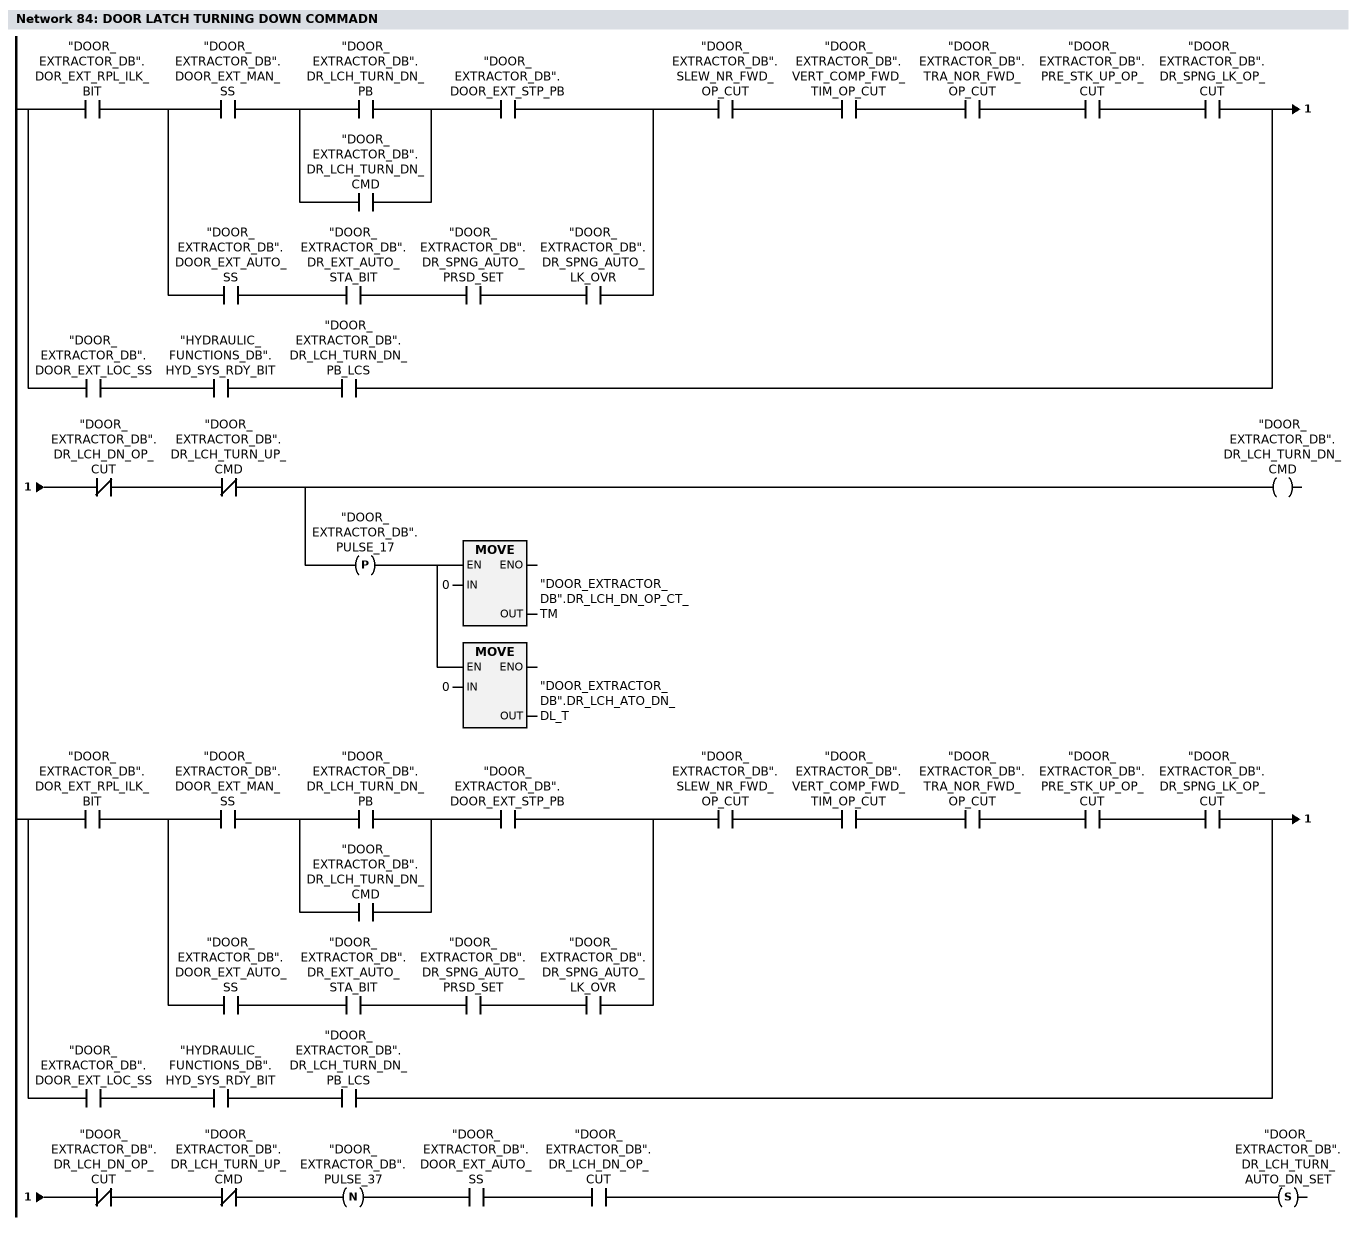
NETWORK
TITLE = DOOR LATCH TURNING DOWN COMMADN
      A(;
      A     "DOOR_EXTRACTOR_DB".DOR_EXT_RPL_ILK_BIT;
      A(;
      A     "DOOR_EXTRACTOR_DB".DOOR_EXT_MAN_SS;
      A(;
      O     "DOOR_EXTRACTOR_DB".DR_LCH_TURN_DN_PB;
      O     "DOOR_EXTRACTOR_DB".DR_LCH_TURN_DN_CMD;
      );
      A     "DOOR_EXTRACTOR_DB".DOOR_EXT_STP_PB;
      O;
      A     "DOOR_EXTRACTOR_DB".DOOR_EXT_AUTO_SS;
      A     "DOOR_EXTRACTOR_DB".DR_EXT_AUTO_STA_BIT;
      A     "DOOR_EXTRACTOR_DB".DR_SPNG_AUTO_PRSD_SET;
      A     "DOOR_EXTRACTOR_DB".DR_SPNG_AUTO_LK_OVR;
      );
      A     "DOOR_EXTRACTOR_DB".SLEW_NR_FWD_OP_CUT;
      A     "DOOR_EXTRACTOR_DB".VERT_COMP_FWD_TIM_OP_CUT;
      A     "DOOR_EXTRACTOR_DB".TRA_NOR_FWD_OP_CUT;
      A     "DOOR_EXTRACTOR_DB".PRE_STK_UP_OP_CUT;
      A     "DOOR_EXTRACTOR_DB".DR_SPNG_LK_OP_CUT;
      O;
      A     "DOOR_EXTRACTOR_DB".DOOR_EXT_LOC_SS;
      A     "HYDRAULIC_FUNCTIONS_DB".HYD_SYS_RDY_BIT;
      A     "DOOR_EXTRACTOR_DB".DR_LCH_TURN_DN_PB_LCS;
      );
      AN    "DOOR_EXTRACTOR_DB".DR_LCH_DN_OP_CUT;
      AN    "DOOR_EXTRACTOR_DB".DR_LCH_TURN_UP_CMD;
      =     L 0.0;
      A     L 0.0;
      BLD   102;
      =     "DOOR_EXTRACTOR_DB".DR_LCH_TURN_DN_CMD;
      A(;
      A     L 0.0;
      FN    "DOOR_EXTRACTOR_DB".PULSE_37;
      );
      A     "DOOR_EXTRACTOR_DB".DOOR_EXT_AUTO_SS;
      A     "DOOR_EXTRACTOR_DB".DR_LCH_DN_OP_CUT;
      S     "DOOR_EXTRACTOR_DB".DR_LCH_TURN_AUTO_DN_SET;
      A     L 0.0;
      FP    "DOOR_EXTRACTOR_DB".PULSE_17;
      =     L 0.1;
      A     L 0.1;
      JNB   _04b;
      L     0;
      T     "DOOR_EXTRACTOR_DB".DR_LCH_DN_OP_CT_TM;
_04b: NOP   0;
      A     L 0.1;
      JNB   _04c;
      L     0;
      T     "DOOR_EXTRACTOR_DB".DR_LCH_ATO_DN_DL_T;
_04c: NOP   0;
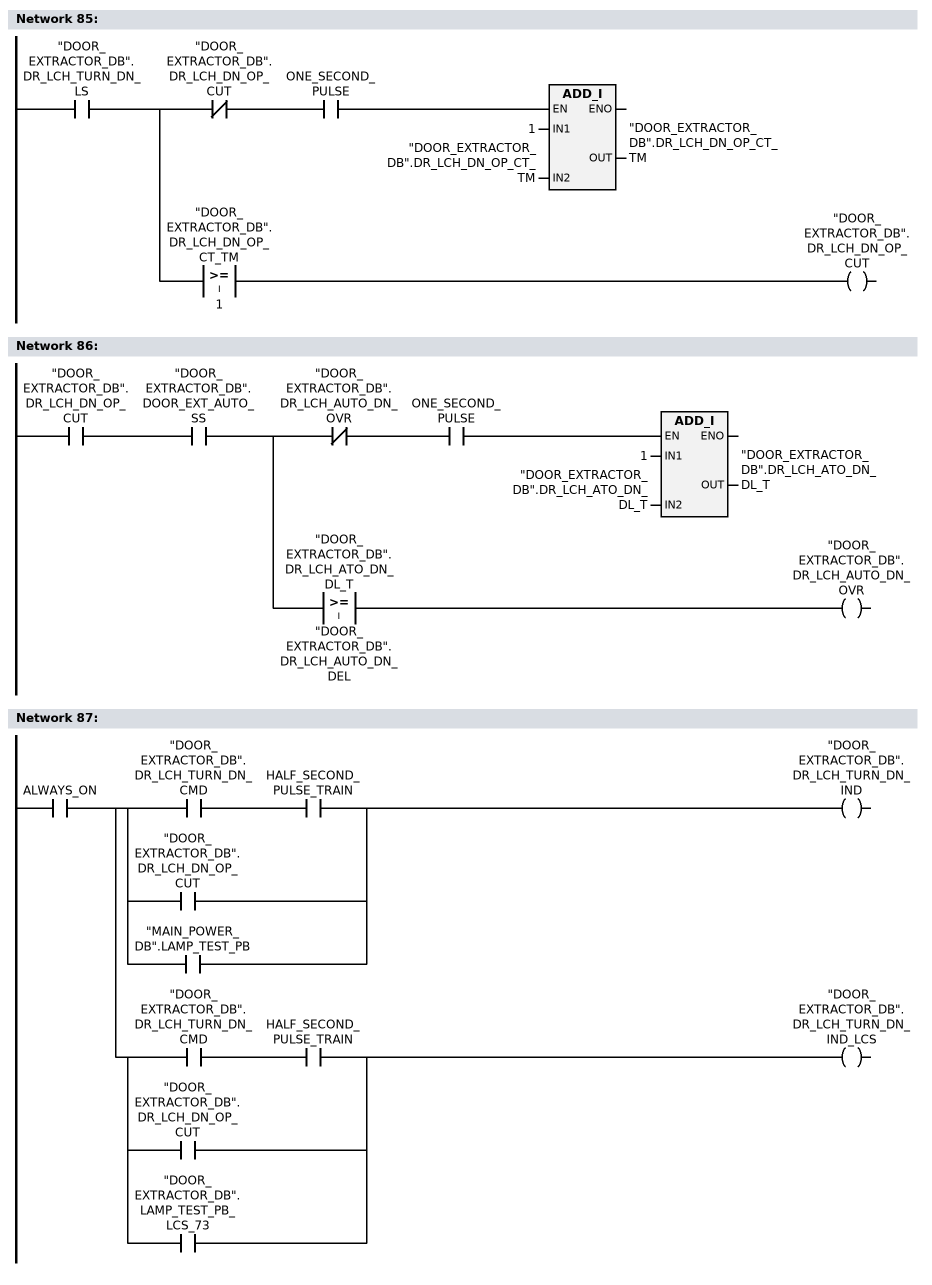
NETWORK
TITLE =
      A     "DOOR_EXTRACTOR_DB".DR_LCH_TURN_DN_LS;
      =     L 0.0;
      A     L 0.0;
      AN    "DOOR_EXTRACTOR_DB".DR_LCH_DN_OP_CUT;
      A     "ONE_SECOND_PULSE";
      JNB   _04d;
      L     1;
      L     "DOOR_EXTRACTOR_DB".DR_LCH_DN_OP_CT_TM;
      +I;
      T     "DOOR_EXTRACTOR_DB".DR_LCH_DN_OP_CT_TM;
_04d: NOP   0;
      A     L 0.0;
      A(;
      L     "DOOR_EXTRACTOR_DB".DR_LCH_DN_OP_CT_TM;
      L     1;
      >=I;
      );
      =     "DOOR_EXTRACTOR_DB".DR_LCH_DN_OP_CUT;
NETWORK
TITLE =
      A     "DOOR_EXTRACTOR_DB".DR_LCH_DN_OP_CUT;
      A     "DOOR_EXTRACTOR_DB".DOOR_EXT_AUTO_SS;
      =     L 0.0;
      A     L 0.0;
      AN    "DOOR_EXTRACTOR_DB".DR_LCH_AUTO_DN_OVR;
      A     "ONE_SECOND_PULSE";
      JNB   _04e;
      L     1;
      L     "DOOR_EXTRACTOR_DB".DR_LCH_ATO_DN_DL_T;
      +I;
      T     "DOOR_EXTRACTOR_DB".DR_LCH_ATO_DN_DL_T;
_04e: NOP   0;
      A     L 0.0;
      A(;
      L     "DOOR_EXTRACTOR_DB".DR_LCH_ATO_DN_DL_T;
      L     "DOOR_EXTRACTOR_DB".DR_LCH_AUTO_DN_DEL;
      >=I;
      );
      =     "DOOR_EXTRACTOR_DB".DR_LCH_AUTO_DN_OVR;
NETWORK
TITLE =
      A     "ALWAYS_ON";
      =     L 0.0;
      A     L 0.0;
      A(;
      A     "DOOR_EXTRACTOR_DB".DR_LCH_TURN_DN_CMD;
      A     "HALF_SECOND_PULSE_TRAIN";
      O     "DOOR_EXTRACTOR_DB".DR_LCH_DN_OP_CUT;
      O     "MAIN_POWER_DB".LAMP_TEST_PB;
      );
      =     "DOOR_EXTRACTOR_DB".DR_LCH_TURN_DN_IND;
      A     L 0.0;
      A(;
      A     "DOOR_EXTRACTOR_DB".DR_LCH_TURN_DN_CMD;
      A     "HALF_SECOND_PULSE_TRAIN";
      O     "DOOR_EXTRACTOR_DB".DR_LCH_DN_OP_CUT;
      O     "DOOR_EXTRACTOR_DB".LAMP_TEST_PB_LCS_73;
      );
      =     "DOOR_EXTRACTOR_DB".DR_LCH_TURN_DN_IND_LCS;
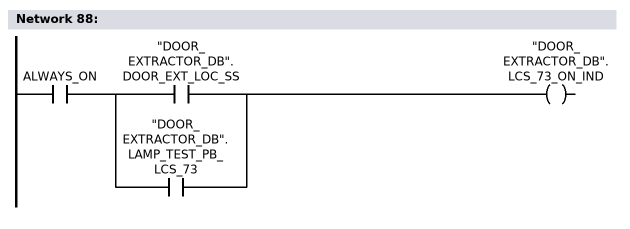
NETWORK
TITLE =
      A     "ALWAYS_ON";
      A(;
      O     "DOOR_EXTRACTOR_DB".DOOR_EXT_LOC_SS;
      O     "DOOR_EXTRACTOR_DB".LAMP_TEST_PB_LCS_73;
      );
      =     "DOOR_EXTRACTOR_DB".LCS_73_ON_IND;
END_FUNCTION

FUNCTION "DOOR_CLEANER" : VOID	// FC 15
AUTHOR : Kamillas
VERSION : 0.1
BEGIN
// (block stored without names or comments; labels and parameter names are numbered)
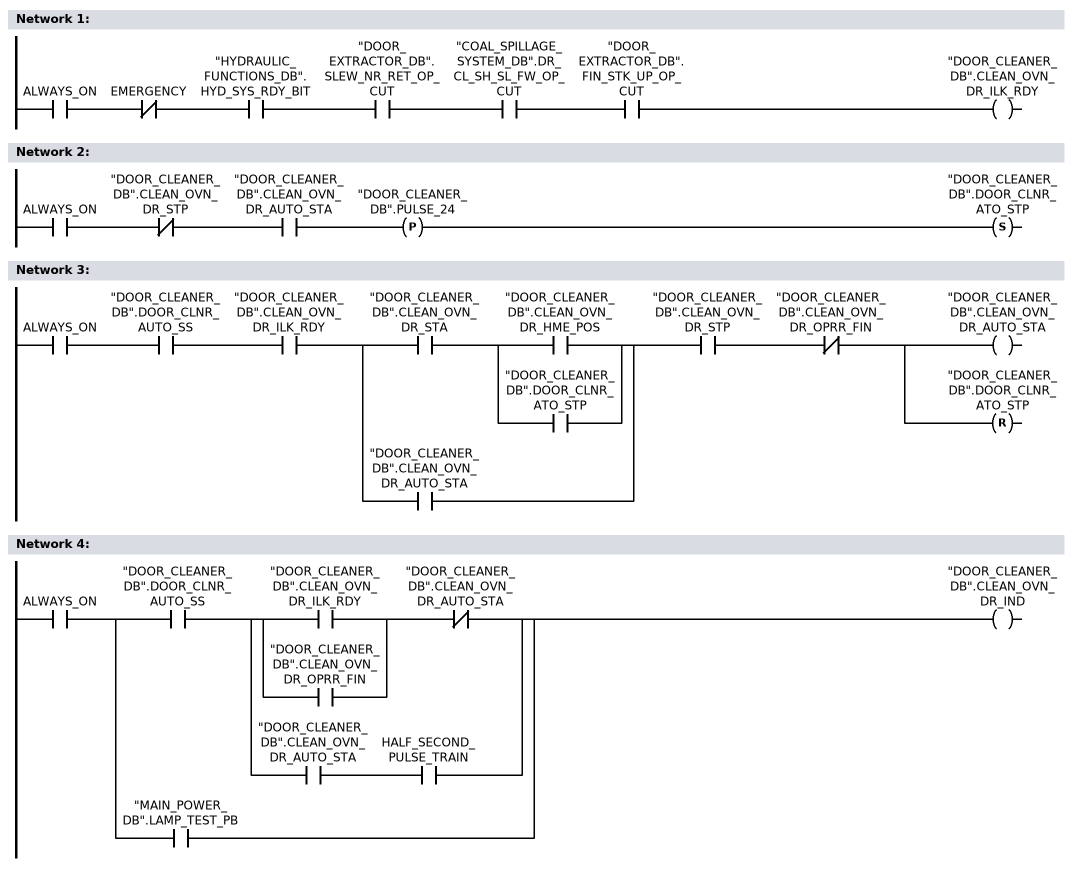
NETWORK
TITLE =
      A     "ALWAYS_ON";
      AN    "EMERGENCY";
      A     "HYDRAULIC_FUNCTIONS_DB".HYD_SYS_RDY_BIT;
      A     "DOOR_EXTRACTOR_DB".SLEW_NR_RET_OP_CUT;
      A     "COAL_SPILLAGE_SYSTEM_DB".DR_CL_SH_SL_FW_OP_CUT;
      A     "DOOR_EXTRACTOR_DB".FIN_STK_UP_OP_CUT;
      =     "DOOR_CLEANER_DB".CLEAN_OVN_DR_ILK_RDY;
NETWORK
TITLE =
      A     "ALWAYS_ON";
      AN    "DOOR_CLEANER_DB".CLEAN_OVN_DR_STP;
      A     "DOOR_CLEANER_DB".CLEAN_OVN_DR_AUTO_STA;
      FP    "DOOR_CLEANER_DB".PULSE_24;
      S     "DOOR_CLEANER_DB".DOOR_CLNR_ATO_STP;
NETWORK
TITLE =
      A     "ALWAYS_ON";
      A     "DOOR_CLEANER_DB".DOOR_CLNR_AUTO_SS;
      A     "DOOR_CLEANER_DB".CLEAN_OVN_DR_ILK_RDY;
      A(;
      A     "DOOR_CLEANER_DB".CLEAN_OVN_DR_STA;
      A(;
      O     "DOOR_CLEANER_DB".CLEAN_OVN_DR_HME_POS;
      O     "DOOR_CLEANER_DB".DOOR_CLNR_ATO_STP;
      );
      O     "DOOR_CLEANER_DB".CLEAN_OVN_DR_AUTO_STA;
      );
      A     "DOOR_CLEANER_DB".CLEAN_OVN_DR_STP;
      AN    "DOOR_CLEANER_DB".CLEAN_OVN_DR_OPRR_FIN;
      =     "DOOR_CLEANER_DB".CLEAN_OVN_DR_AUTO_STA;
      R     "DOOR_CLEANER_DB".DOOR_CLNR_ATO_STP;
NETWORK
TITLE =
      A     "ALWAYS_ON";
      A(;
      A     "DOOR_CLEANER_DB".DOOR_CLNR_AUTO_SS;
      A(;
      A(;
      O     "DOOR_CLEANER_DB".CLEAN_OVN_DR_ILK_RDY;
      O     "DOOR_CLEANER_DB".CLEAN_OVN_DR_OPRR_FIN;
      );
      AN    "DOOR_CLEANER_DB".CLEAN_OVN_DR_AUTO_STA;
      O;
      A     "DOOR_CLEANER_DB".CLEAN_OVN_DR_AUTO_STA;
      A     "HALF_SECOND_PULSE_TRAIN";
      );
      O     "MAIN_POWER_DB".LAMP_TEST_PB;
      );
      =     "DOOR_CLEANER_DB".CLEAN_OVN_DR_IND;
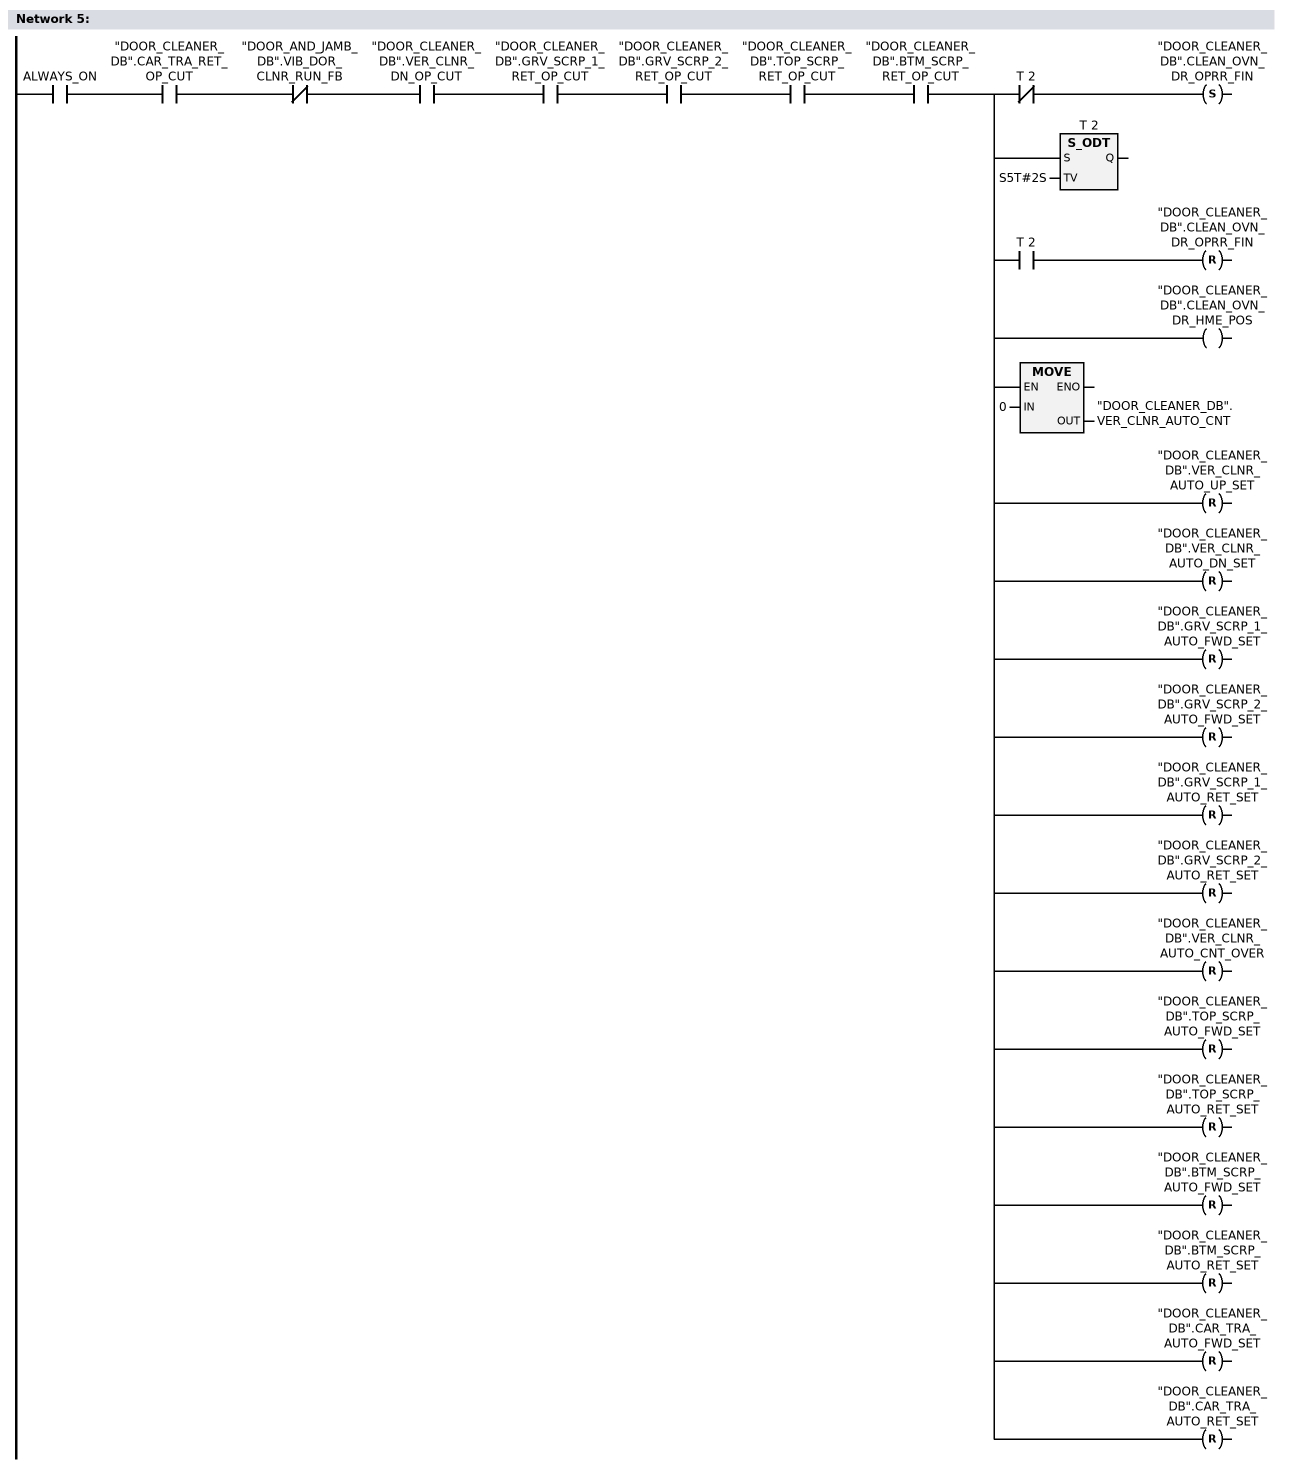
NETWORK
TITLE =
      A     "ALWAYS_ON";
      A     "DOOR_CLEANER_DB".CAR_TRA_RET_OP_CUT;
      AN    "DOOR_AND_JAMB_DB".VIB_DOR_CLNR_RUN_FB;
      A     "DOOR_CLEANER_DB".VER_CLNR_DN_OP_CUT;
      A     "DOOR_CLEANER_DB".GRV_SCRP_1_RET_OP_CUT;
      A     "DOOR_CLEANER_DB".GRV_SCRP_2_RET_OP_CUT;
      A     "DOOR_CLEANER_DB".TOP_SCRP_RET_OP_CUT;
      A     "DOOR_CLEANER_DB".BTM_SCRP_RET_OP_CUT;
      =     L 0.0;
      A     L 0.0;
      AN    T 2;
      S     "DOOR_CLEANER_DB".CLEAN_OVN_DR_OPRR_FIN;
      A     L 0.0;
      L     S5T#2S;
      SD    T 2;
      NOP   0;
      NOP   0;
      NOP   0;
      NOP   0;
      A     L 0.0;
      A     T 2;
      R     "DOOR_CLEANER_DB".CLEAN_OVN_DR_OPRR_FIN;
      A     L 0.0;
      BLD   102;
      =     "DOOR_CLEANER_DB".CLEAN_OVN_DR_HME_POS;
      A     L 0.0;
      JNB   M001;
      L     0;
      T     "DOOR_CLEANER_DB".VER_CLNR_AUTO_CNT;
M001: NOP   0;
      A     L 0.0;
      BLD   102;
      R     "DOOR_CLEANER_DB".VER_CLNR_AUTO_UP_SET;
      A     L 0.0;
      BLD   102;
      R     "DOOR_CLEANER_DB".VER_CLNR_AUTO_DN_SET;
      A     L 0.0;
      BLD   102;
      R     "DOOR_CLEANER_DB".GRV_SCRP_1_AUTO_FWD_SET;
      A     L 0.0;
      BLD   102;
      R     "DOOR_CLEANER_DB".GRV_SCRP_2_AUTO_FWD_SET;
      A     L 0.0;
      BLD   102;
      R     "DOOR_CLEANER_DB".GRV_SCRP_1_AUTO_RET_SET;
      A     L 0.0;
      BLD   102;
      R     "DOOR_CLEANER_DB".GRV_SCRP_2_AUTO_RET_SET;
      A     L 0.0;
      BLD   102;
      R     "DOOR_CLEANER_DB".VER_CLNR_AUTO_CNT_OVER;
      A     L 0.0;
      BLD   102;
      R     "DOOR_CLEANER_DB".TOP_SCRP_AUTO_FWD_SET;
      A     L 0.0;
      BLD   102;
      R     "DOOR_CLEANER_DB".TOP_SCRP_AUTO_RET_SET;
      A     L 0.0;
      BLD   102;
      R     "DOOR_CLEANER_DB".BTM_SCRP_AUTO_FWD_SET;
      A     L 0.0;
      BLD   102;
      R     "DOOR_CLEANER_DB".BTM_SCRP_AUTO_RET_SET;
      A     L 0.0;
      BLD   102;
      R     "DOOR_CLEANER_DB".CAR_TRA_AUTO_FWD_SET;
      A     L 0.0;
      BLD   102;
      R     "DOOR_CLEANER_DB".CAR_TRA_AUTO_RET_SET;
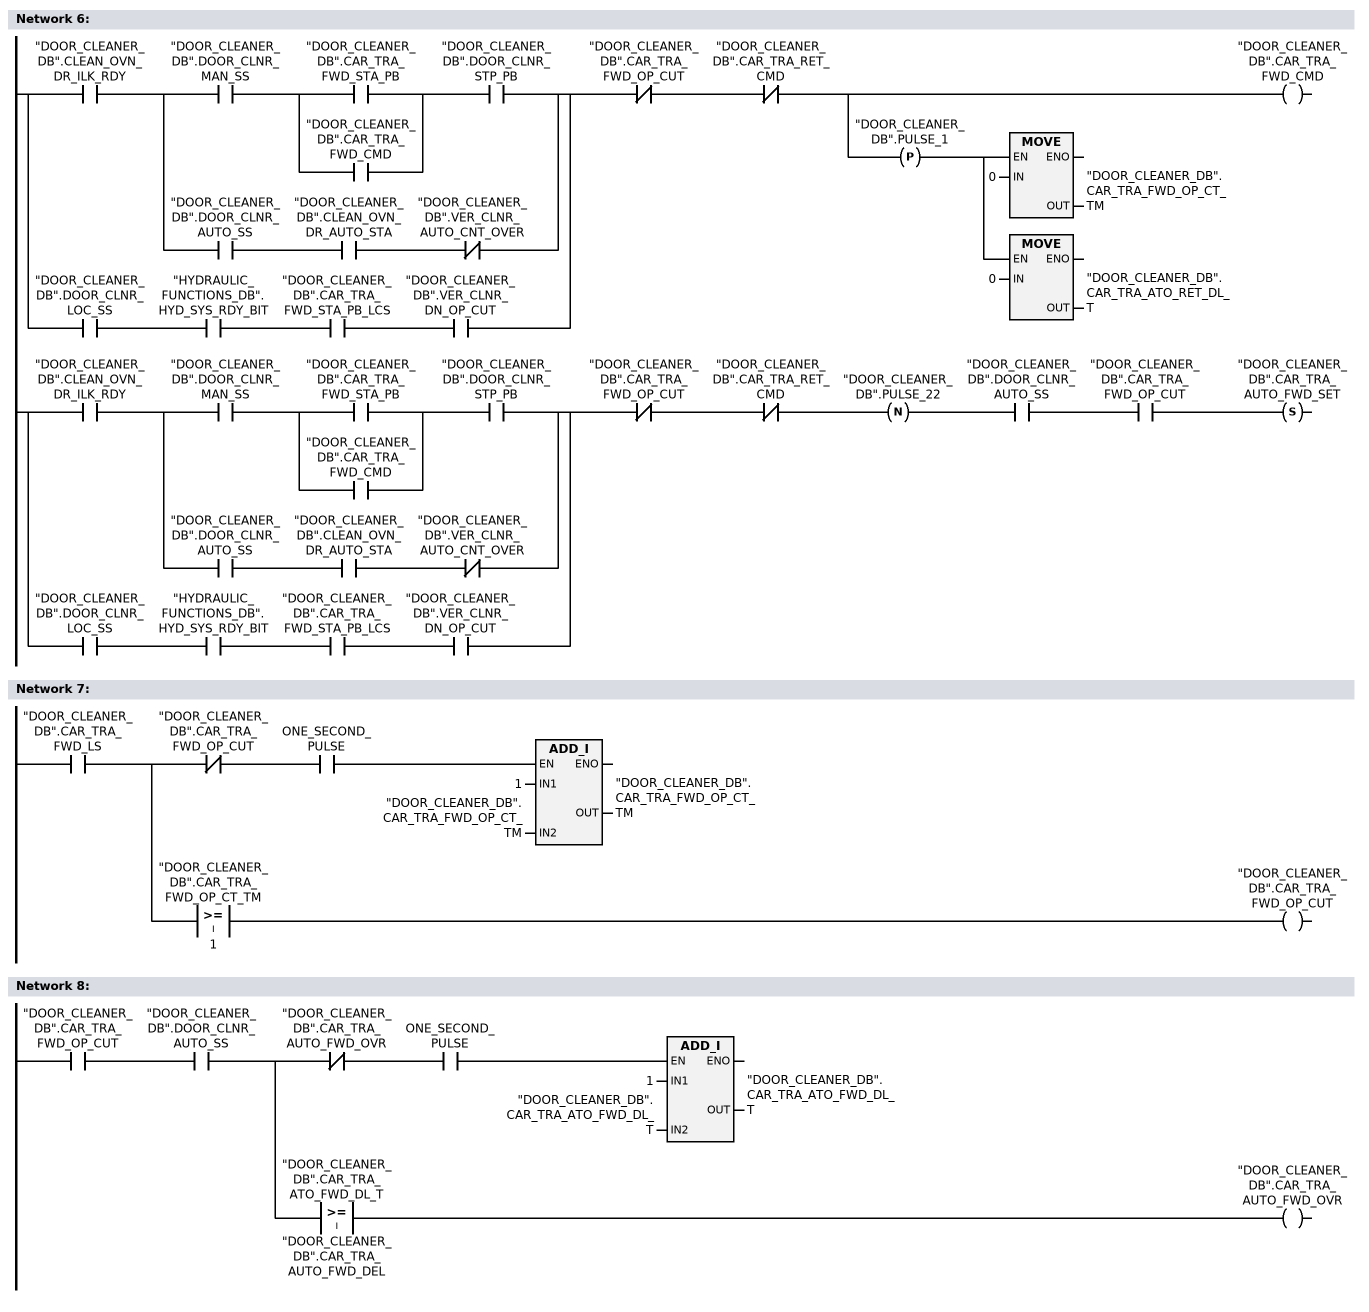
NETWORK
TITLE =
      A(;
      A     "DOOR_CLEANER_DB".CLEAN_OVN_DR_ILK_RDY;
      A(;
      A     "DOOR_CLEANER_DB".DOOR_CLNR_MAN_SS;
      A(;
      O     "DOOR_CLEANER_DB".CAR_TRA_FWD_STA_PB;
      O     "DOOR_CLEANER_DB".CAR_TRA_FWD_CMD;
      );
      A     "DOOR_CLEANER_DB".DOOR_CLNR_STP_PB;
      O;
      A     "DOOR_CLEANER_DB".DOOR_CLNR_AUTO_SS;
      A     "DOOR_CLEANER_DB".CLEAN_OVN_DR_AUTO_STA;
      AN    "DOOR_CLEANER_DB".VER_CLNR_AUTO_CNT_OVER;
      );
      O;
      A     "DOOR_CLEANER_DB".DOOR_CLNR_LOC_SS;
      A     "HYDRAULIC_FUNCTIONS_DB".HYD_SYS_RDY_BIT;
      A     "DOOR_CLEANER_DB".CAR_TRA_FWD_STA_PB_LCS;
      A     "DOOR_CLEANER_DB".VER_CLNR_DN_OP_CUT;
      );
      AN    "DOOR_CLEANER_DB".CAR_TRA_FWD_OP_CUT;
      AN    "DOOR_CLEANER_DB".CAR_TRA_RET_CMD;
      =     L 0.0;
      A     L 0.0;
      BLD   102;
      =     "DOOR_CLEANER_DB".CAR_TRA_FWD_CMD;
      A(;
      A     L 0.0;
      FN    "DOOR_CLEANER_DB".PULSE_22;
      );
      A     "DOOR_CLEANER_DB".DOOR_CLNR_AUTO_SS;
      A     "DOOR_CLEANER_DB".CAR_TRA_FWD_OP_CUT;
      S     "DOOR_CLEANER_DB".CAR_TRA_AUTO_FWD_SET;
      A     L 0.0;
      FP    "DOOR_CLEANER_DB".PULSE_1;
      =     L 0.1;
      A     L 0.1;
      JNB   M002;
      L     0;
      T     "DOOR_CLEANER_DB".CAR_TRA_FWD_OP_CT_TM;
M002: NOP   0;
      A     L 0.1;
      JNB   M003;
      L     0;
      T     "DOOR_CLEANER_DB".CAR_TRA_ATO_RET_DL_T;
M003: NOP   0;
NETWORK
TITLE =
      A     "DOOR_CLEANER_DB".CAR_TRA_FWD_LS;
      =     L 0.0;
      A     L 0.0;
      AN    "DOOR_CLEANER_DB".CAR_TRA_FWD_OP_CUT;
      A     "ONE_SECOND_PULSE";
      JNB   M004;
      L     1;
      L     "DOOR_CLEANER_DB".CAR_TRA_FWD_OP_CT_TM;
      +I;
      T     "DOOR_CLEANER_DB".CAR_TRA_FWD_OP_CT_TM;
M004: NOP   0;
      A     L 0.0;
      A(;
      L     "DOOR_CLEANER_DB".CAR_TRA_FWD_OP_CT_TM;
      L     1;
      >=I;
      );
      =     "DOOR_CLEANER_DB".CAR_TRA_FWD_OP_CUT;
NETWORK
TITLE =
      A     "DOOR_CLEANER_DB".CAR_TRA_FWD_OP_CUT;
      A     "DOOR_CLEANER_DB".DOOR_CLNR_AUTO_SS;
      =     L 0.0;
      A     L 0.0;
      AN    "DOOR_CLEANER_DB".CAR_TRA_AUTO_FWD_OVR;
      A     "ONE_SECOND_PULSE";
      JNB   M005;
      L     1;
      L     "DOOR_CLEANER_DB".CAR_TRA_ATO_FWD_DL_T;
      +I;
      T     "DOOR_CLEANER_DB".CAR_TRA_ATO_FWD_DL_T;
M005: NOP   0;
      A     L 0.0;
      A(;
      L     "DOOR_CLEANER_DB".CAR_TRA_ATO_FWD_DL_T;
      L     "DOOR_CLEANER_DB".CAR_TRA_AUTO_FWD_DEL;
      >=I;
      );
      =     "DOOR_CLEANER_DB".CAR_TRA_AUTO_FWD_OVR;
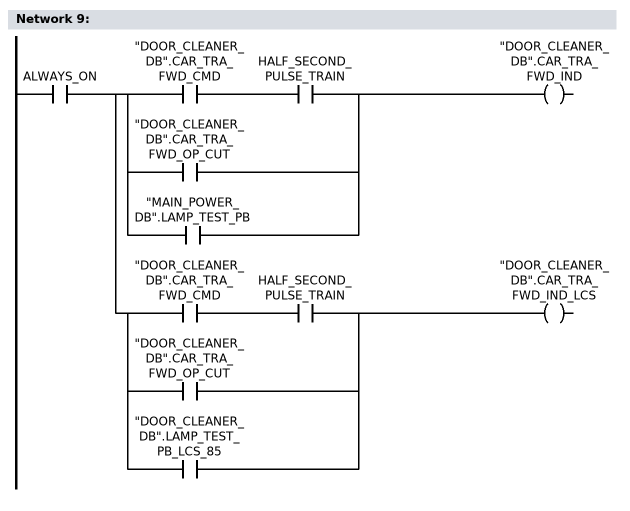
NETWORK
TITLE =
      A     "ALWAYS_ON";
      =     L 0.0;
      A     L 0.0;
      A(;
      A     "DOOR_CLEANER_DB".CAR_TRA_FWD_CMD;
      A     "HALF_SECOND_PULSE_TRAIN";
      O     "DOOR_CLEANER_DB".CAR_TRA_FWD_OP_CUT;
      O     "MAIN_POWER_DB".LAMP_TEST_PB;
      );
      =     "DOOR_CLEANER_DB".CAR_TRA_FWD_IND;
      A     L 0.0;
      A(;
      A     "DOOR_CLEANER_DB".CAR_TRA_FWD_CMD;
      A     "HALF_SECOND_PULSE_TRAIN";
      O     "DOOR_CLEANER_DB".CAR_TRA_FWD_OP_CUT;
      O     "DOOR_CLEANER_DB".LAMP_TEST_PB_LCS_85;
      );
      =     "DOOR_CLEANER_DB".CAR_TRA_FWD_IND_LCS;
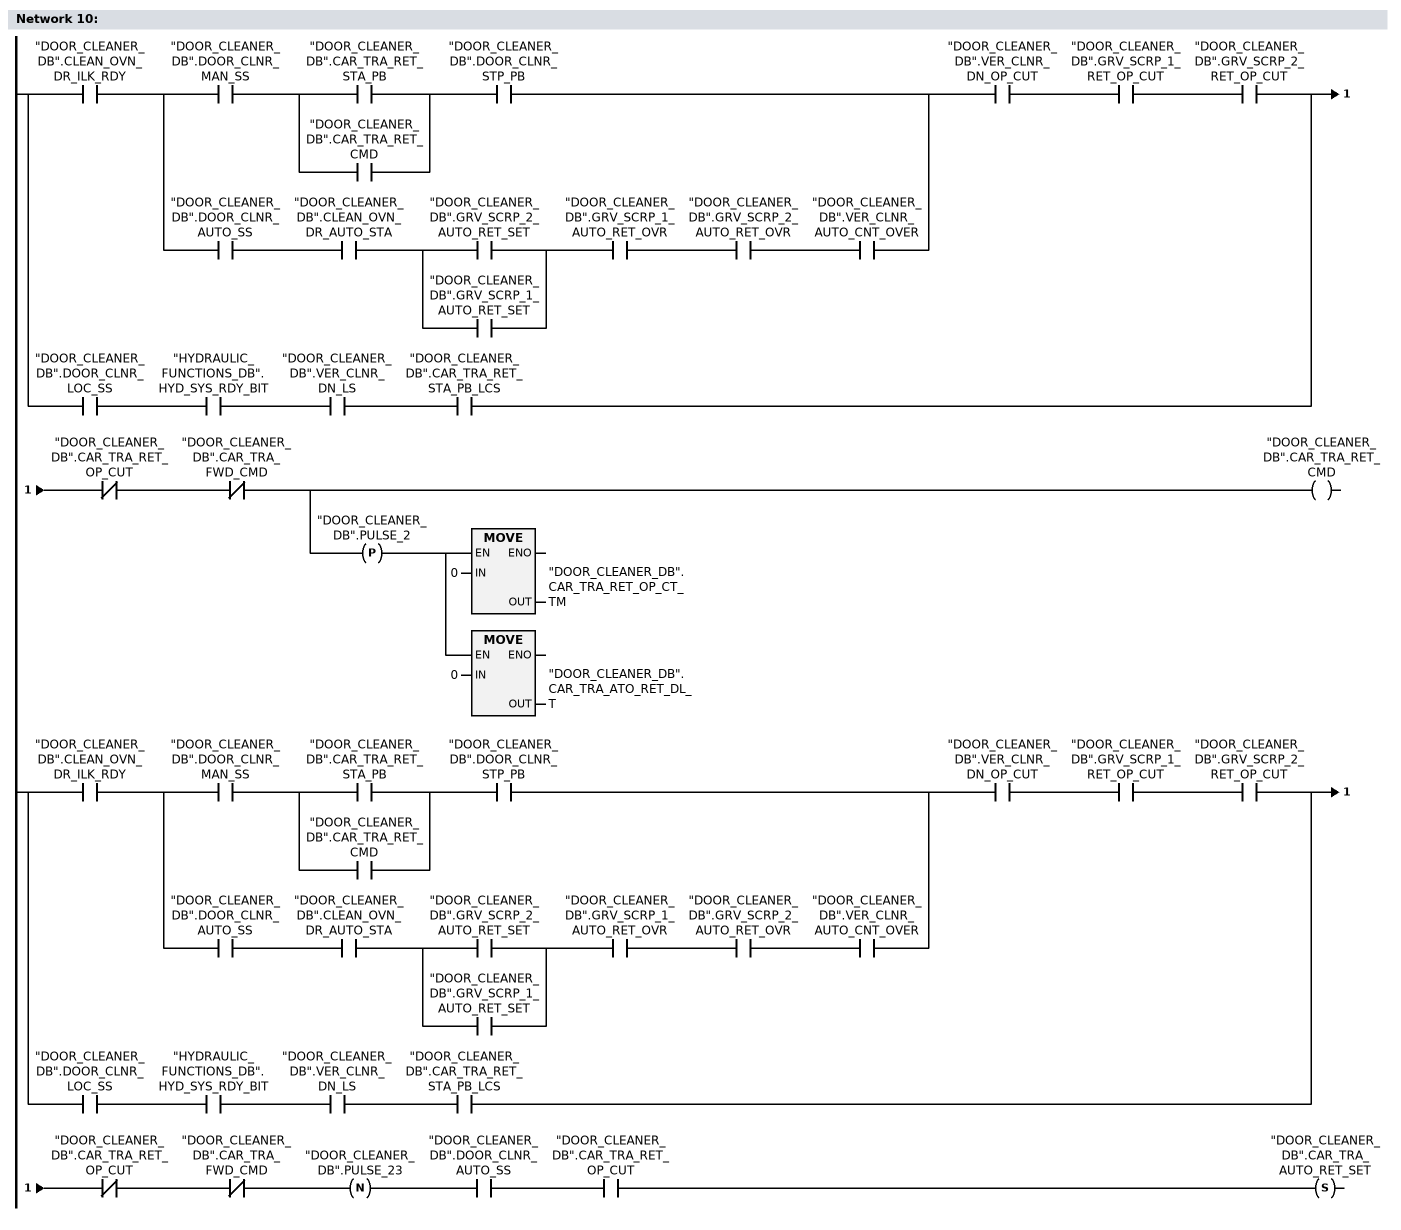
NETWORK
TITLE =
      A(;
      A     "DOOR_CLEANER_DB".CLEAN_OVN_DR_ILK_RDY;
      A(;
      A     "DOOR_CLEANER_DB".DOOR_CLNR_MAN_SS;
      A(;
      O     "DOOR_CLEANER_DB".CAR_TRA_RET_STA_PB;
      O     "DOOR_CLEANER_DB".CAR_TRA_RET_CMD;
      );
      A     "DOOR_CLEANER_DB".DOOR_CLNR_STP_PB;
      O;
      A     "DOOR_CLEANER_DB".DOOR_CLNR_AUTO_SS;
      A     "DOOR_CLEANER_DB".CLEAN_OVN_DR_AUTO_STA;
      A(;
      O     "DOOR_CLEANER_DB".GRV_SCRP_2_AUTO_RET_SET;
      O     "DOOR_CLEANER_DB".GRV_SCRP_1_AUTO_RET_SET;
      );
      A     "DOOR_CLEANER_DB".GRV_SCRP_1_AUTO_RET_OVR;
      A     "DOOR_CLEANER_DB".GRV_SCRP_2_AUTO_RET_OVR;
      A     "DOOR_CLEANER_DB".VER_CLNR_AUTO_CNT_OVER;
      );
      A     "DOOR_CLEANER_DB".VER_CLNR_DN_OP_CUT;
      A     "DOOR_CLEANER_DB".GRV_SCRP_1_RET_OP_CUT;
      A     "DOOR_CLEANER_DB".GRV_SCRP_2_RET_OP_CUT;
      O;
      A     "DOOR_CLEANER_DB".DOOR_CLNR_LOC_SS;
      A     "HYDRAULIC_FUNCTIONS_DB".HYD_SYS_RDY_BIT;
      A     "DOOR_CLEANER_DB".VER_CLNR_DN_LS;
      A     "DOOR_CLEANER_DB".CAR_TRA_RET_STA_PB_LCS;
      );
      AN    "DOOR_CLEANER_DB".CAR_TRA_RET_OP_CUT;
      AN    "DOOR_CLEANER_DB".CAR_TRA_FWD_CMD;
      =     L 0.0;
      A     L 0.0;
      BLD   102;
      =     "DOOR_CLEANER_DB".CAR_TRA_RET_CMD;
      A(;
      A     L 0.0;
      FN    "DOOR_CLEANER_DB".PULSE_23;
      );
      A     "DOOR_CLEANER_DB".DOOR_CLNR_AUTO_SS;
      A     "DOOR_CLEANER_DB".CAR_TRA_RET_OP_CUT;
      S     "DOOR_CLEANER_DB".CAR_TRA_AUTO_RET_SET;
      A     L 0.0;
      FP    "DOOR_CLEANER_DB".PULSE_2;
      =     L 0.1;
      A     L 0.1;
      JNB   M006;
      L     0;
      T     "DOOR_CLEANER_DB".CAR_TRA_RET_OP_CT_TM;
M006: NOP   0;
      A     L 0.1;
      JNB   M007;
      L     0;
      T     "DOOR_CLEANER_DB".CAR_TRA_ATO_RET_DL_T;
M007: NOP   0;
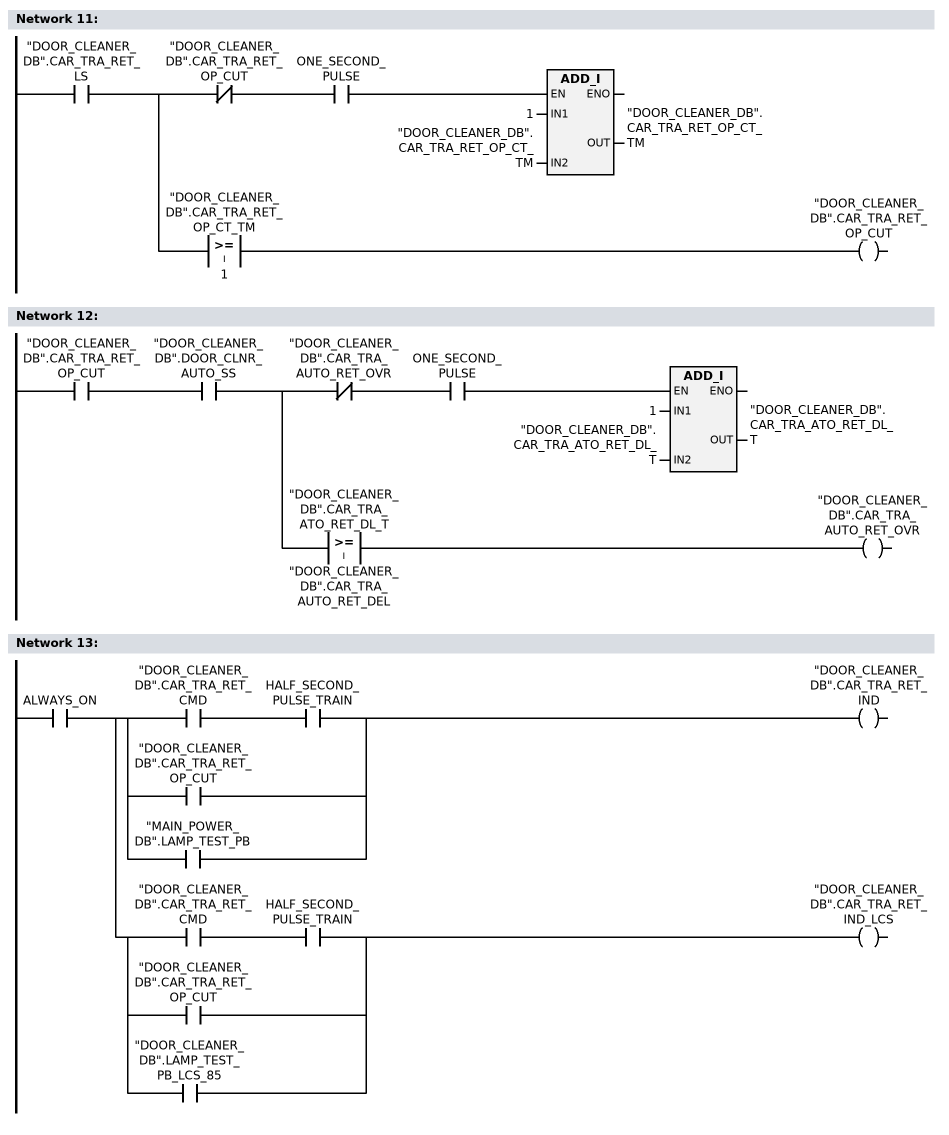
NETWORK
TITLE =
      A     "DOOR_CLEANER_DB".CAR_TRA_RET_LS;
      =     L 0.0;
      A     L 0.0;
      AN    "DOOR_CLEANER_DB".CAR_TRA_RET_OP_CUT;
      A     "ONE_SECOND_PULSE";
      JNB   M008;
      L     1;
      L     "DOOR_CLEANER_DB".CAR_TRA_RET_OP_CT_TM;
      +I;
      T     "DOOR_CLEANER_DB".CAR_TRA_RET_OP_CT_TM;
M008: NOP   0;
      A     L 0.0;
      A(;
      L     "DOOR_CLEANER_DB".CAR_TRA_RET_OP_CT_TM;
      L     1;
      >=I;
      );
      =     "DOOR_CLEANER_DB".CAR_TRA_RET_OP_CUT;
NETWORK
TITLE =
      A     "DOOR_CLEANER_DB".CAR_TRA_RET_OP_CUT;
      A     "DOOR_CLEANER_DB".DOOR_CLNR_AUTO_SS;
      =     L 0.0;
      A     L 0.0;
      AN    "DOOR_CLEANER_DB".CAR_TRA_AUTO_RET_OVR;
      A     "ONE_SECOND_PULSE";
      JNB   M009;
      L     1;
      L     "DOOR_CLEANER_DB".CAR_TRA_ATO_RET_DL_T;
      +I;
      T     "DOOR_CLEANER_DB".CAR_TRA_ATO_RET_DL_T;
M009: NOP   0;
      A     L 0.0;
      A(;
      L     "DOOR_CLEANER_DB".CAR_TRA_ATO_RET_DL_T;
      L     "DOOR_CLEANER_DB".CAR_TRA_AUTO_RET_DEL;
      >=I;
      );
      =     "DOOR_CLEANER_DB".CAR_TRA_AUTO_RET_OVR;
NETWORK
TITLE =
      A     "ALWAYS_ON";
      =     L 0.0;
      A     L 0.0;
      A(;
      A     "DOOR_CLEANER_DB".CAR_TRA_RET_CMD;
      A     "HALF_SECOND_PULSE_TRAIN";
      O     "DOOR_CLEANER_DB".CAR_TRA_RET_OP_CUT;
      O     "MAIN_POWER_DB".LAMP_TEST_PB;
      );
      =     "DOOR_CLEANER_DB".CAR_TRA_RET_IND;
      A     L 0.0;
      A(;
      A     "DOOR_CLEANER_DB".CAR_TRA_RET_CMD;
      A     "HALF_SECOND_PULSE_TRAIN";
      O     "DOOR_CLEANER_DB".CAR_TRA_RET_OP_CUT;
      O     "DOOR_CLEANER_DB".LAMP_TEST_PB_LCS_85;
      );
      =     "DOOR_CLEANER_DB".CAR_TRA_RET_IND_LCS;
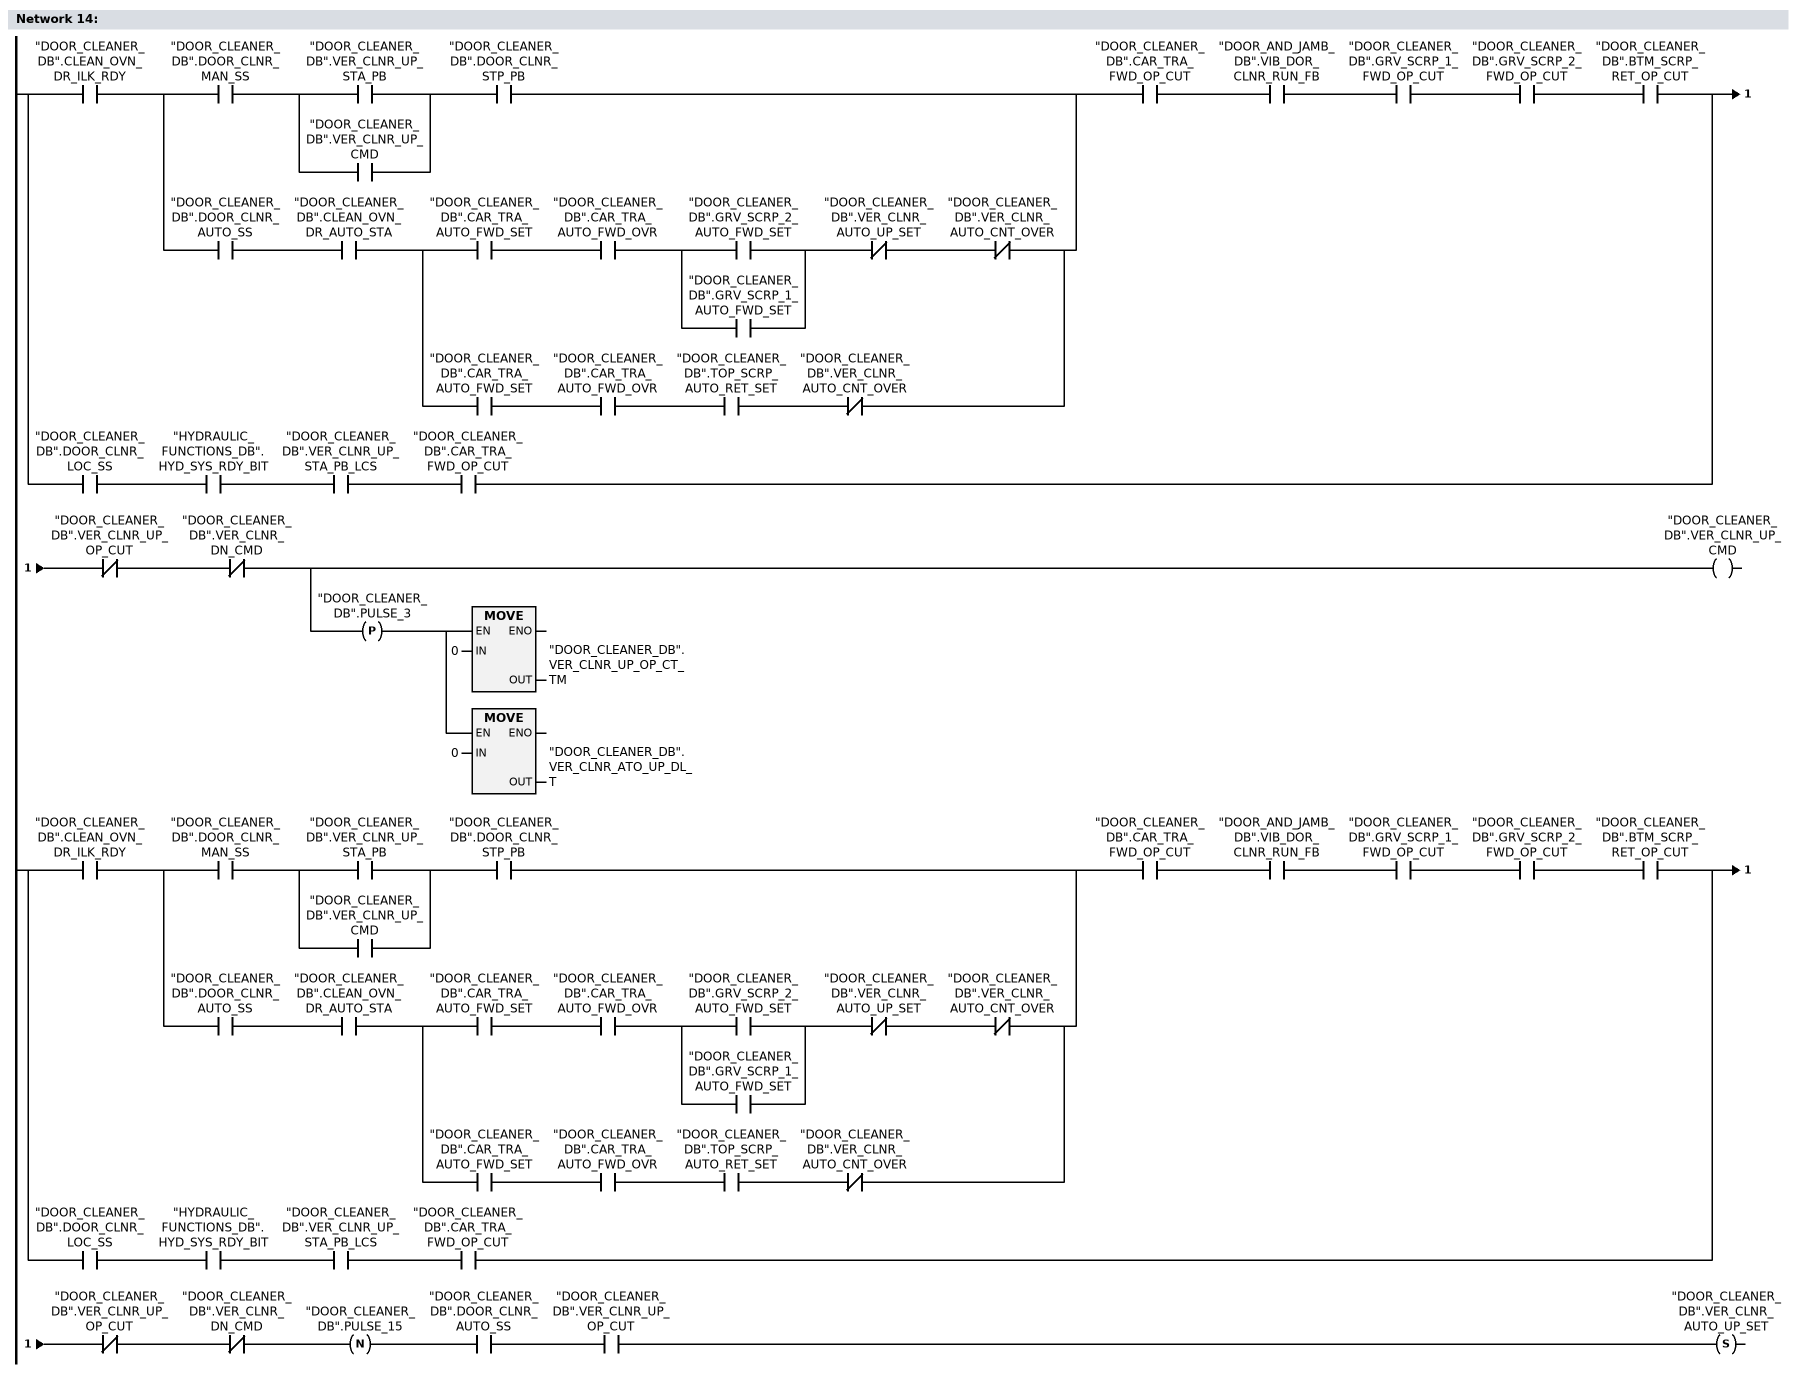
NETWORK
TITLE =
      A(;
      A     "DOOR_CLEANER_DB".CLEAN_OVN_DR_ILK_RDY;
      A(;
      A     "DOOR_CLEANER_DB".DOOR_CLNR_MAN_SS;
      A(;
      O     "DOOR_CLEANER_DB".VER_CLNR_UP_STA_PB;
      O     "DOOR_CLEANER_DB".VER_CLNR_UP_CMD;
      );
      A     "DOOR_CLEANER_DB".DOOR_CLNR_STP_PB;
      O;
      A     "DOOR_CLEANER_DB".DOOR_CLNR_AUTO_SS;
      A     "DOOR_CLEANER_DB".CLEAN_OVN_DR_AUTO_STA;
      A(;
      A     "DOOR_CLEANER_DB".CAR_TRA_AUTO_FWD_SET;
      A     "DOOR_CLEANER_DB".CAR_TRA_AUTO_FWD_OVR;
      A(;
      O     "DOOR_CLEANER_DB".GRV_SCRP_2_AUTO_FWD_SET;
      O     "DOOR_CLEANER_DB".GRV_SCRP_1_AUTO_FWD_SET;
      );
      AN    "DOOR_CLEANER_DB".VER_CLNR_AUTO_UP_SET;
      AN    "DOOR_CLEANER_DB".VER_CLNR_AUTO_CNT_OVER;
      O;
      A     "DOOR_CLEANER_DB".CAR_TRA_AUTO_FWD_SET;
      A     "DOOR_CLEANER_DB".CAR_TRA_AUTO_FWD_OVR;
      A     "DOOR_CLEANER_DB".TOP_SCRP_AUTO_RET_SET;
      AN    "DOOR_CLEANER_DB".VER_CLNR_AUTO_CNT_OVER;
      );
      );
      A     "DOOR_CLEANER_DB".CAR_TRA_FWD_OP_CUT;
      A     "DOOR_AND_JAMB_DB".VIB_DOR_CLNR_RUN_FB;
      A     "DOOR_CLEANER_DB".GRV_SCRP_1_FWD_OP_CUT;
      A     "DOOR_CLEANER_DB".GRV_SCRP_2_FWD_OP_CUT;
      A     "DOOR_CLEANER_DB".BTM_SCRP_RET_OP_CUT;
      O;
      A     "DOOR_CLEANER_DB".DOOR_CLNR_LOC_SS;
      A     "HYDRAULIC_FUNCTIONS_DB".HYD_SYS_RDY_BIT;
      A     "DOOR_CLEANER_DB".VER_CLNR_UP_STA_PB_LCS;
      A     "DOOR_CLEANER_DB".CAR_TRA_FWD_OP_CUT;
      );
      AN    "DOOR_CLEANER_DB".VER_CLNR_UP_OP_CUT;
      AN    "DOOR_CLEANER_DB".VER_CLNR_DN_CMD;
      =     L 0.0;
      A     L 0.0;
      BLD   102;
      =     "DOOR_CLEANER_DB".VER_CLNR_UP_CMD;
      A(;
      A     L 0.0;
      FN    "DOOR_CLEANER_DB".PULSE_15;
      );
      A     "DOOR_CLEANER_DB".DOOR_CLNR_AUTO_SS;
      A     "DOOR_CLEANER_DB".VER_CLNR_UP_OP_CUT;
      S     "DOOR_CLEANER_DB".VER_CLNR_AUTO_UP_SET;
      A     L 0.0;
      FP    "DOOR_CLEANER_DB".PULSE_3;
      =     L 0.1;
      A     L 0.1;
      JNB   M010;
      L     0;
      T     "DOOR_CLEANER_DB".VER_CLNR_UP_OP_CT_TM;
M010: NOP   0;
      A     L 0.1;
      JNB   M011;
      L     0;
      T     "DOOR_CLEANER_DB".VER_CLNR_ATO_UP_DL_T;
M011: NOP   0;
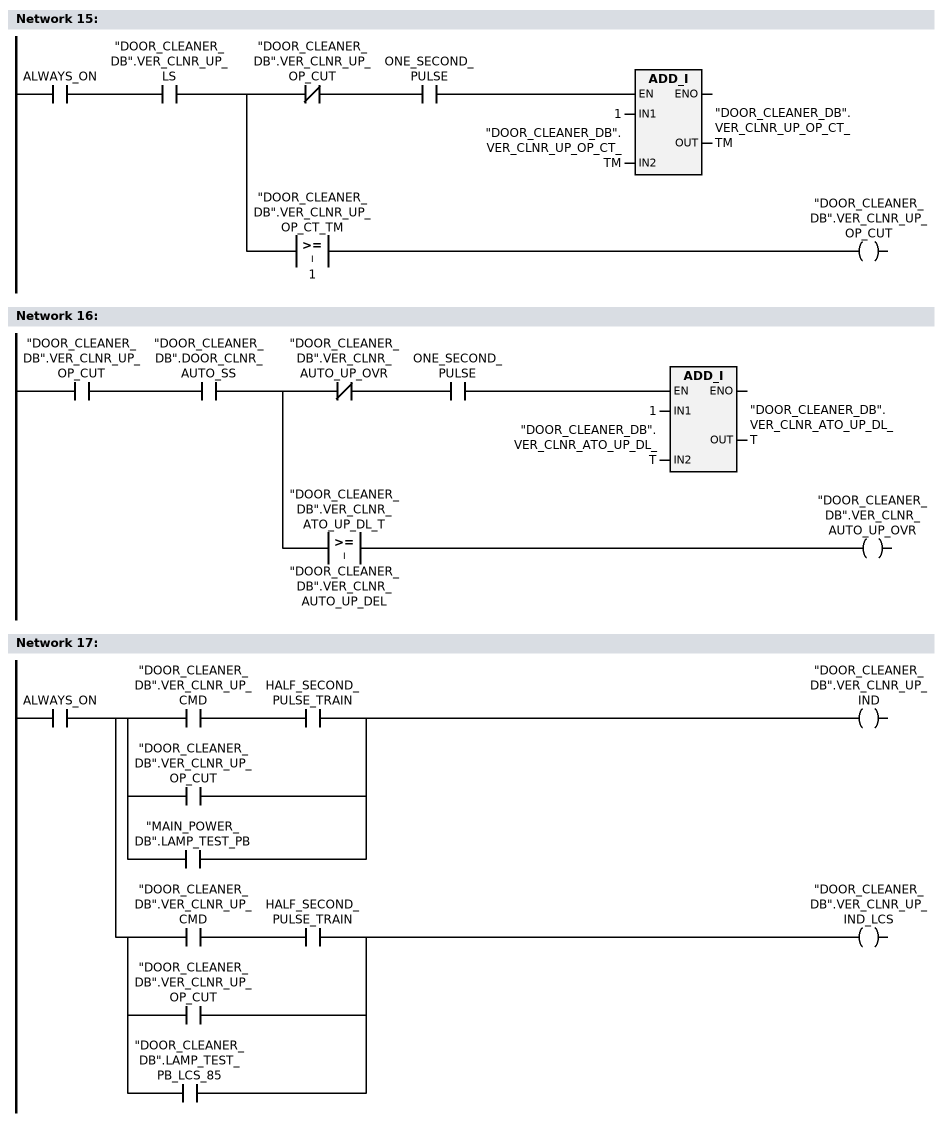
NETWORK
TITLE =
      A     "ALWAYS_ON";
      A     "DOOR_CLEANER_DB".VER_CLNR_UP_LS;
      =     L 0.0;
      A     L 0.0;
      AN    "DOOR_CLEANER_DB".VER_CLNR_UP_OP_CUT;
      A     "ONE_SECOND_PULSE";
      JNB   M012;
      L     1;
      L     "DOOR_CLEANER_DB".VER_CLNR_UP_OP_CT_TM;
      +I;
      T     "DOOR_CLEANER_DB".VER_CLNR_UP_OP_CT_TM;
M012: NOP   0;
      A     L 0.0;
      A(;
      L     "DOOR_CLEANER_DB".VER_CLNR_UP_OP_CT_TM;
      L     1;
      >=I;
      );
      =     "DOOR_CLEANER_DB".VER_CLNR_UP_OP_CUT;
NETWORK
TITLE =
      A     "DOOR_CLEANER_DB".VER_CLNR_UP_OP_CUT;
      A     "DOOR_CLEANER_DB".DOOR_CLNR_AUTO_SS;
      =     L 0.0;
      A     L 0.0;
      AN    "DOOR_CLEANER_DB".VER_CLNR_AUTO_UP_OVR;
      A     "ONE_SECOND_PULSE";
      JNB   M013;
      L     1;
      L     "DOOR_CLEANER_DB".VER_CLNR_ATO_UP_DL_T;
      +I;
      T     "DOOR_CLEANER_DB".VER_CLNR_ATO_UP_DL_T;
M013: NOP   0;
      A     L 0.0;
      A(;
      L     "DOOR_CLEANER_DB".VER_CLNR_ATO_UP_DL_T;
      L     "DOOR_CLEANER_DB".VER_CLNR_AUTO_UP_DEL;
      >=I;
      );
      =     "DOOR_CLEANER_DB".VER_CLNR_AUTO_UP_OVR;
NETWORK
TITLE =
      A     "ALWAYS_ON";
      =     L 0.0;
      A     L 0.0;
      A(;
      A     "DOOR_CLEANER_DB".VER_CLNR_UP_CMD;
      A     "HALF_SECOND_PULSE_TRAIN";
      O     "DOOR_CLEANER_DB".VER_CLNR_UP_OP_CUT;
      O     "MAIN_POWER_DB".LAMP_TEST_PB;
      );
      =     "DOOR_CLEANER_DB".VER_CLNR_UP_IND;
      A     L 0.0;
      A(;
      A     "DOOR_CLEANER_DB".VER_CLNR_UP_CMD;
      A     "HALF_SECOND_PULSE_TRAIN";
      O     "DOOR_CLEANER_DB".VER_CLNR_UP_OP_CUT;
      O     "DOOR_CLEANER_DB".LAMP_TEST_PB_LCS_85;
      );
      =     "DOOR_CLEANER_DB".VER_CLNR_UP_IND_LCS;
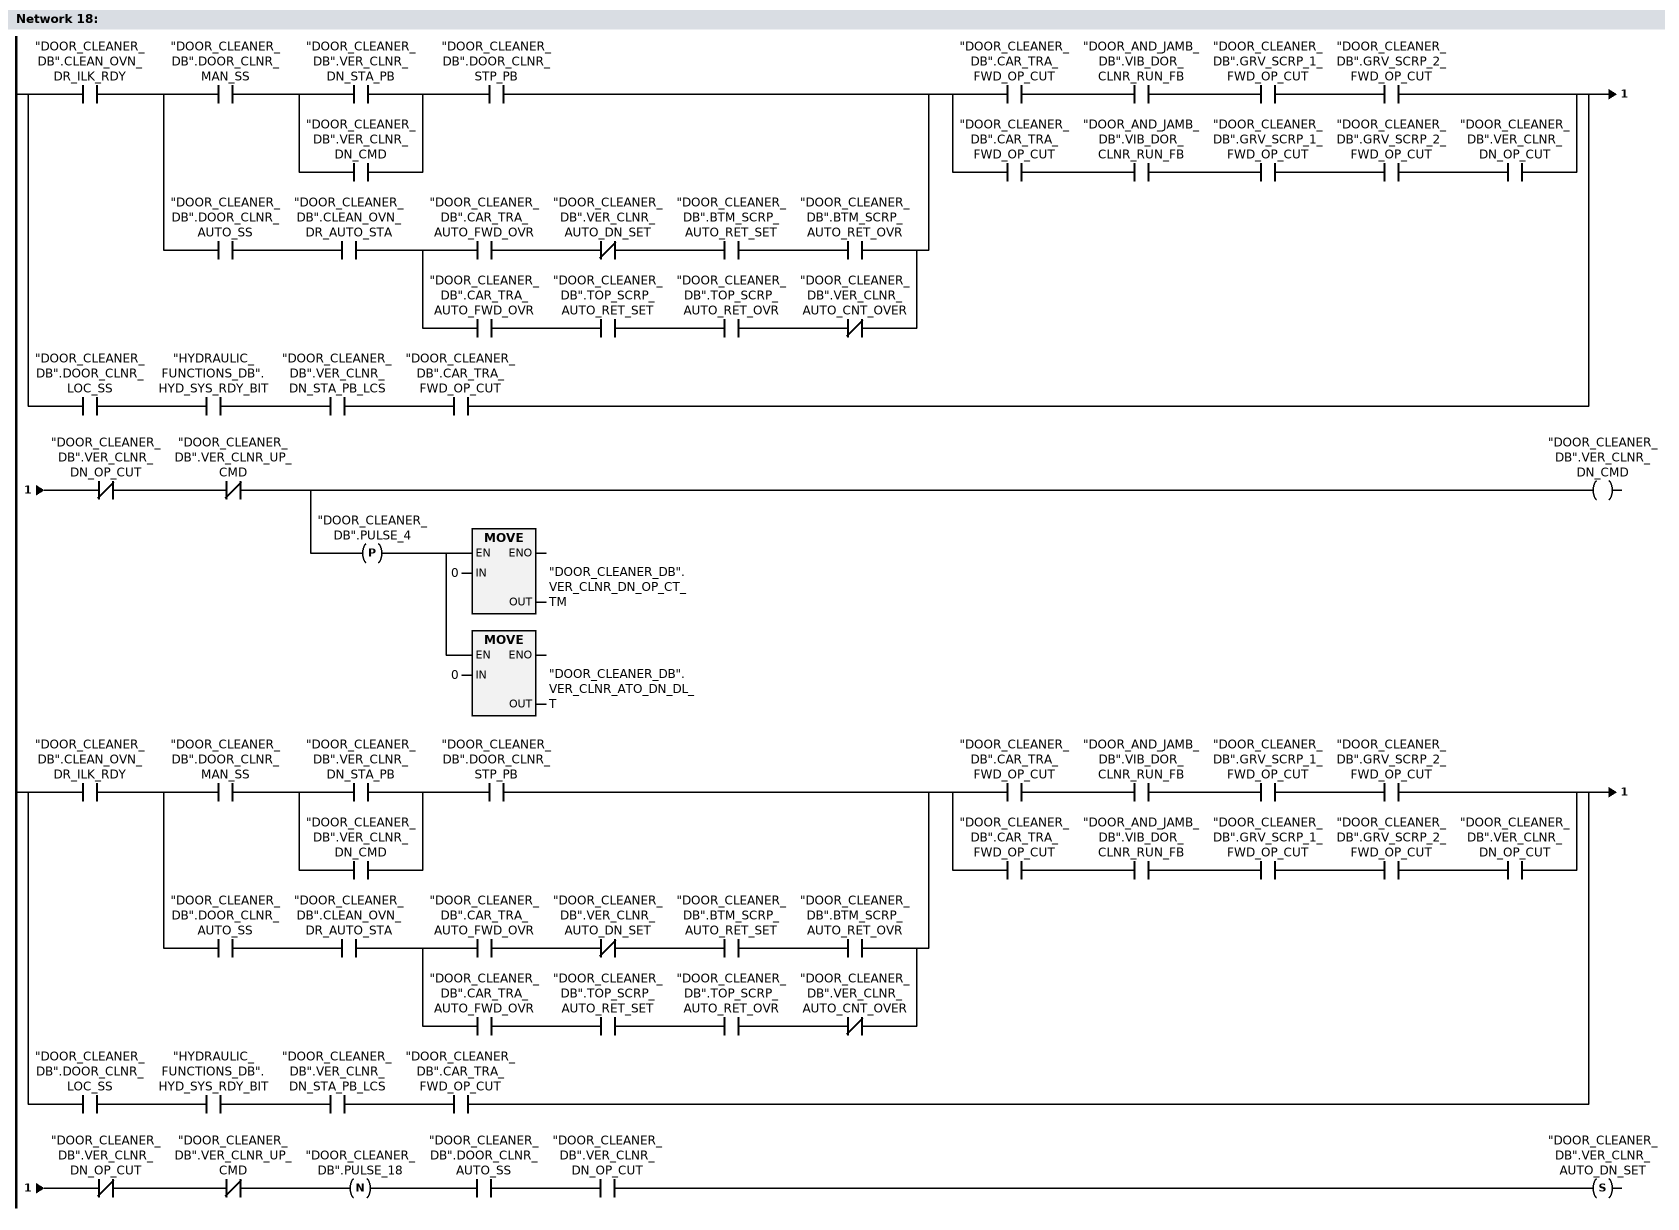
NETWORK
TITLE =
      A(;
      A     "DOOR_CLEANER_DB".CLEAN_OVN_DR_ILK_RDY;
      A(;
      A     "DOOR_CLEANER_DB".DOOR_CLNR_MAN_SS;
      A(;
      O     "DOOR_CLEANER_DB".VER_CLNR_DN_STA_PB;
      O     "DOOR_CLEANER_DB".VER_CLNR_DN_CMD;
      );
      A     "DOOR_CLEANER_DB".DOOR_CLNR_STP_PB;
      O;
      A     "DOOR_CLEANER_DB".DOOR_CLNR_AUTO_SS;
      A     "DOOR_CLEANER_DB".CLEAN_OVN_DR_AUTO_STA;
      A(;
      A     "DOOR_CLEANER_DB".CAR_TRA_AUTO_FWD_OVR;
      AN    "DOOR_CLEANER_DB".VER_CLNR_AUTO_DN_SET;
      A     "DOOR_CLEANER_DB".BTM_SCRP_AUTO_RET_SET;
      A     "DOOR_CLEANER_DB".BTM_SCRP_AUTO_RET_OVR;
      O;
      A     "DOOR_CLEANER_DB".CAR_TRA_AUTO_FWD_OVR;
      A     "DOOR_CLEANER_DB".TOP_SCRP_AUTO_RET_SET;
      A     "DOOR_CLEANER_DB".TOP_SCRP_AUTO_RET_OVR;
      AN    "DOOR_CLEANER_DB".VER_CLNR_AUTO_CNT_OVER;
      );
      );
      A(;
      A     "DOOR_CLEANER_DB".CAR_TRA_FWD_OP_CUT;
      A     "DOOR_AND_JAMB_DB".VIB_DOR_CLNR_RUN_FB;
      A     "DOOR_CLEANER_DB".GRV_SCRP_1_FWD_OP_CUT;
      A     "DOOR_CLEANER_DB".GRV_SCRP_2_FWD_OP_CUT;
      O;
      A     "DOOR_CLEANER_DB".CAR_TRA_FWD_OP_CUT;
      A     "DOOR_AND_JAMB_DB".VIB_DOR_CLNR_RUN_FB;
      A     "DOOR_CLEANER_DB".GRV_SCRP_1_FWD_OP_CUT;
      A     "DOOR_CLEANER_DB".GRV_SCRP_2_FWD_OP_CUT;
      A     "DOOR_CLEANER_DB".VER_CLNR_DN_OP_CUT;
      );
      O;
      A     "DOOR_CLEANER_DB".DOOR_CLNR_LOC_SS;
      A     "HYDRAULIC_FUNCTIONS_DB".HYD_SYS_RDY_BIT;
      A     "DOOR_CLEANER_DB".VER_CLNR_DN_STA_PB_LCS;
      A     "DOOR_CLEANER_DB".CAR_TRA_FWD_OP_CUT;
      );
      AN    "DOOR_CLEANER_DB".VER_CLNR_DN_OP_CUT;
      AN    "DOOR_CLEANER_DB".VER_CLNR_UP_CMD;
      =     L 0.0;
      A     L 0.0;
      BLD   102;
      =     "DOOR_CLEANER_DB".VER_CLNR_DN_CMD;
      A(;
      A     L 0.0;
      FN    "DOOR_CLEANER_DB".PULSE_18;
      );
      A     "DOOR_CLEANER_DB".DOOR_CLNR_AUTO_SS;
      A     "DOOR_CLEANER_DB".VER_CLNR_DN_OP_CUT;
      S     "DOOR_CLEANER_DB".VER_CLNR_AUTO_DN_SET;
      A     L 0.0;
      FP    "DOOR_CLEANER_DB".PULSE_4;
      =     L 0.1;
      A     L 0.1;
      JNB   M014;
      L     0;
      T     "DOOR_CLEANER_DB".VER_CLNR_DN_OP_CT_TM;
M014: NOP   0;
      A     L 0.1;
      JNB   M015;
      L     0;
      T     "DOOR_CLEANER_DB".VER_CLNR_ATO_DN_DL_T;
M015: NOP   0;
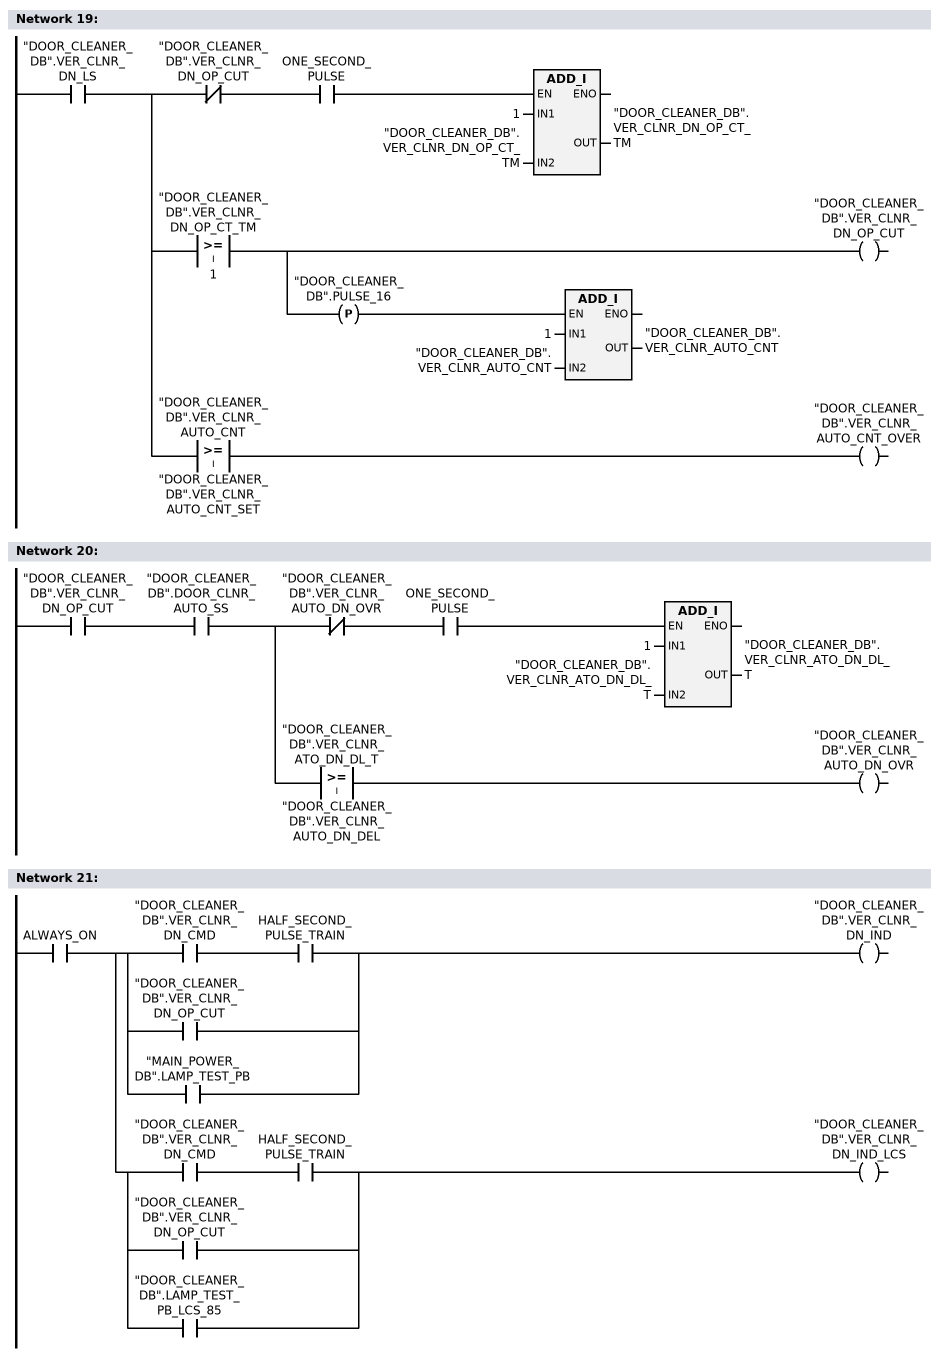
NETWORK
TITLE =
      A     "DOOR_CLEANER_DB".VER_CLNR_DN_LS;
      =     L 0.0;
      A     L 0.0;
      AN    "DOOR_CLEANER_DB".VER_CLNR_DN_OP_CUT;
      A     "ONE_SECOND_PULSE";
      JNB   M016;
      L     1;
      L     "DOOR_CLEANER_DB".VER_CLNR_DN_OP_CT_TM;
      +I;
      T     "DOOR_CLEANER_DB".VER_CLNR_DN_OP_CT_TM;
M016: NOP   0;
      A     L 0.0;
      A(;
      L     "DOOR_CLEANER_DB".VER_CLNR_DN_OP_CT_TM;
      L     1;
      >=I;
      );
      =     L 0.1;
      A     L 0.1;
      BLD   102;
      =     "DOOR_CLEANER_DB".VER_CLNR_DN_OP_CUT;
      A     L 0.1;
      FP    "DOOR_CLEANER_DB".PULSE_16;
      JNB   M017;
      L     1;
      L     "DOOR_CLEANER_DB".VER_CLNR_AUTO_CNT;
      +I;
      T     "DOOR_CLEANER_DB".VER_CLNR_AUTO_CNT;
M017: NOP   0;
      A     L 0.0;
      A(;
      L     "DOOR_CLEANER_DB".VER_CLNR_AUTO_CNT;
      L     "DOOR_CLEANER_DB".VER_CLNR_AUTO_CNT_SET;
      >=I;
      );
      =     "DOOR_CLEANER_DB".VER_CLNR_AUTO_CNT_OVER;
NETWORK
TITLE =
      A     "DOOR_CLEANER_DB".VER_CLNR_DN_OP_CUT;
      A     "DOOR_CLEANER_DB".DOOR_CLNR_AUTO_SS;
      =     L 0.0;
      A     L 0.0;
      AN    "DOOR_CLEANER_DB".VER_CLNR_AUTO_DN_OVR;
      A     "ONE_SECOND_PULSE";
      JNB   M018;
      L     1;
      L     "DOOR_CLEANER_DB".VER_CLNR_ATO_DN_DL_T;
      +I;
      T     "DOOR_CLEANER_DB".VER_CLNR_ATO_DN_DL_T;
M018: NOP   0;
      A     L 0.0;
      A(;
      L     "DOOR_CLEANER_DB".VER_CLNR_ATO_DN_DL_T;
      L     "DOOR_CLEANER_DB".VER_CLNR_AUTO_DN_DEL;
      >=I;
      );
      =     "DOOR_CLEANER_DB".VER_CLNR_AUTO_DN_OVR;
NETWORK
TITLE =
      A     "ALWAYS_ON";
      =     L 0.0;
      A     L 0.0;
      A(;
      A     "DOOR_CLEANER_DB".VER_CLNR_DN_CMD;
      A     "HALF_SECOND_PULSE_TRAIN";
      O     "DOOR_CLEANER_DB".VER_CLNR_DN_OP_CUT;
      O     "MAIN_POWER_DB".LAMP_TEST_PB;
      );
      =     "DOOR_CLEANER_DB".VER_CLNR_DN_IND;
      A     L 0.0;
      A(;
      A     "DOOR_CLEANER_DB".VER_CLNR_DN_CMD;
      A     "HALF_SECOND_PULSE_TRAIN";
      O     "DOOR_CLEANER_DB".VER_CLNR_DN_OP_CUT;
      O     "DOOR_CLEANER_DB".LAMP_TEST_PB_LCS_85;
      );
      =     "DOOR_CLEANER_DB".VER_CLNR_DN_IND_LCS;
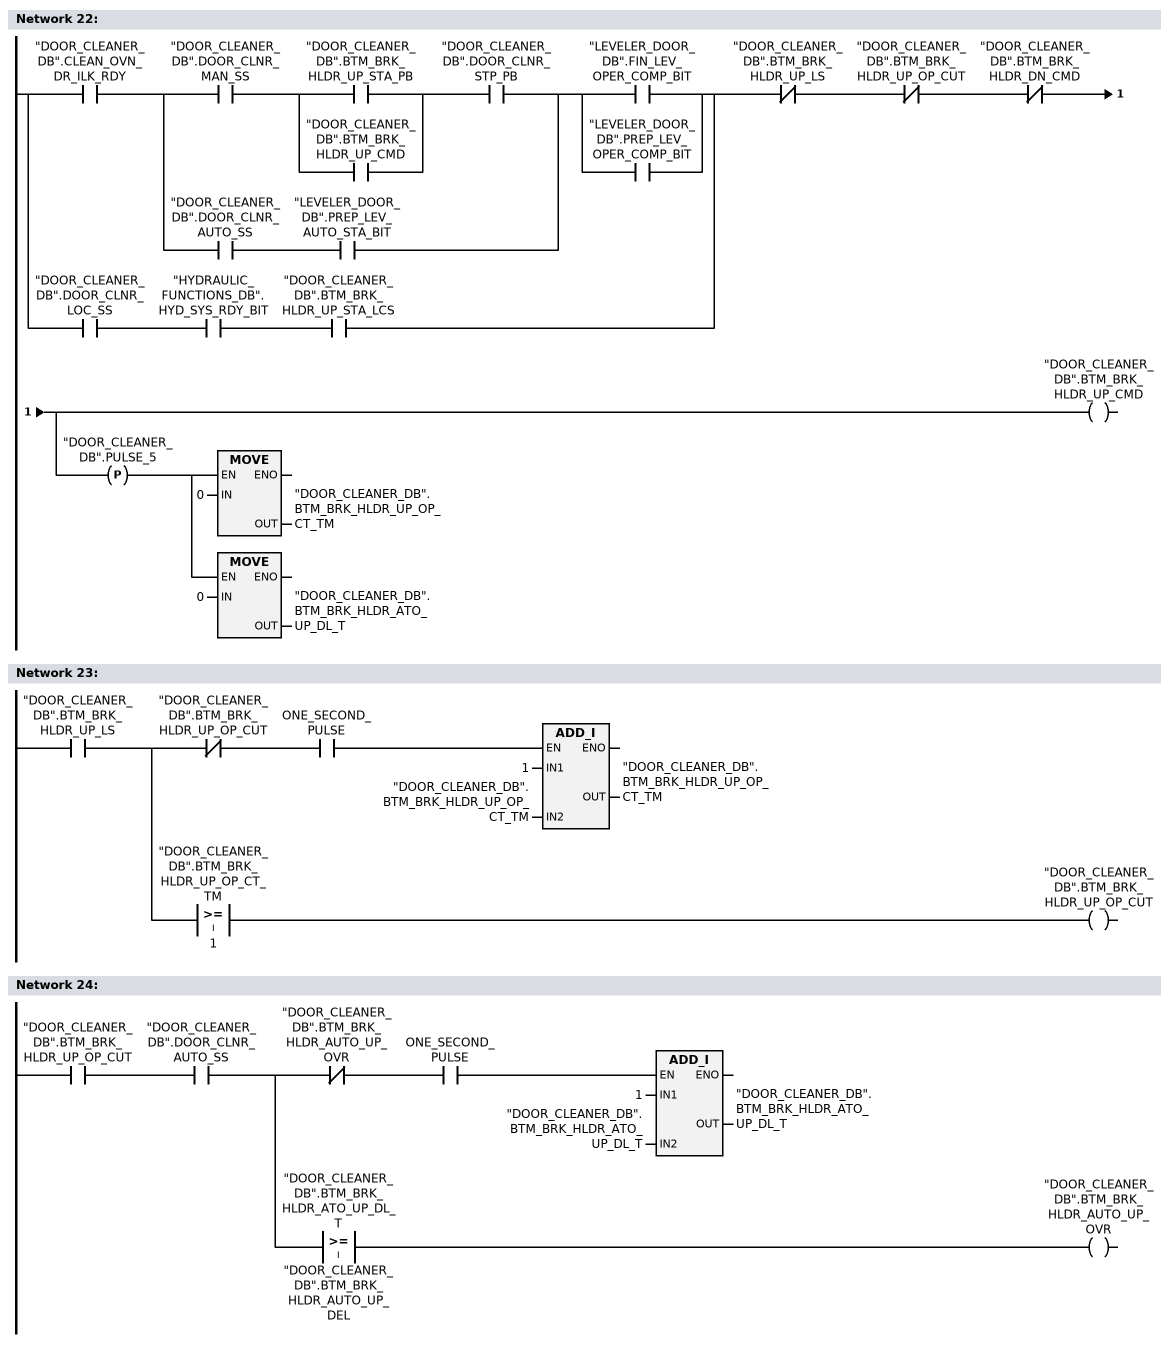
NETWORK
TITLE =
      A(;
      A     "DOOR_CLEANER_DB".CLEAN_OVN_DR_ILK_RDY;
      A(;
      A     "DOOR_CLEANER_DB".DOOR_CLNR_MAN_SS;
      A(;
      O     "DOOR_CLEANER_DB".BTM_BRK_HLDR_UP_STA_PB;
      O     "DOOR_CLEANER_DB".BTM_BRK_HLDR_UP_CMD;
      );
      A     "DOOR_CLEANER_DB".DOOR_CLNR_STP_PB;
      O;
      A     "DOOR_CLEANER_DB".DOOR_CLNR_AUTO_SS;
      A     "LEVELER_DOOR_DB".PREP_LEV_AUTO_STA_BIT;
      );
      A(;
      O     "LEVELER_DOOR_DB".FIN_LEV_OPER_COMP_BIT;
      O     "LEVELER_DOOR_DB".PREP_LEV_OPER_COMP_BIT;
      );
      O;
      A     "DOOR_CLEANER_DB".DOOR_CLNR_LOC_SS;
      A     "HYDRAULIC_FUNCTIONS_DB".HYD_SYS_RDY_BIT;
      A     "DOOR_CLEANER_DB".BTM_BRK_HLDR_UP_STA_LCS;
      );
      AN    "DOOR_CLEANER_DB".BTM_BRK_HLDR_UP_LS;
      AN    "DOOR_CLEANER_DB".BTM_BRK_HLDR_UP_OP_CUT;
      AN    "DOOR_CLEANER_DB".BTM_BRK_HLDR_DN_CMD;
      =     L 0.0;
      A     L 0.0;
      BLD   102;
      =     "DOOR_CLEANER_DB".BTM_BRK_HLDR_UP_CMD;
      A     L 0.0;
      FP    "DOOR_CLEANER_DB".PULSE_5;
      =     L 0.1;
      A     L 0.1;
      JNB   M019;
      L     0;
      T     "DOOR_CLEANER_DB".BTM_BRK_HLDR_UP_OP_CT_TM;
M019: NOP   0;
      A     L 0.1;
      JNB   M020;
      L     0;
      T     "DOOR_CLEANER_DB".BTM_BRK_HLDR_ATO_UP_DL_T;
M020: NOP   0;
NETWORK
TITLE =
      A     "DOOR_CLEANER_DB".BTM_BRK_HLDR_UP_LS;
      =     L 0.0;
      A     L 0.0;
      AN    "DOOR_CLEANER_DB".BTM_BRK_HLDR_UP_OP_CUT;
      A     "ONE_SECOND_PULSE";
      JNB   M021;
      L     1;
      L     "DOOR_CLEANER_DB".BTM_BRK_HLDR_UP_OP_CT_TM;
      +I;
      T     "DOOR_CLEANER_DB".BTM_BRK_HLDR_UP_OP_CT_TM;
M021: NOP   0;
      A     L 0.0;
      A(;
      L     "DOOR_CLEANER_DB".BTM_BRK_HLDR_UP_OP_CT_TM;
      L     1;
      >=I;
      );
      =     "DOOR_CLEANER_DB".BTM_BRK_HLDR_UP_OP_CUT;
NETWORK
TITLE =
      A     "DOOR_CLEANER_DB".BTM_BRK_HLDR_UP_OP_CUT;
      A     "DOOR_CLEANER_DB".DOOR_CLNR_AUTO_SS;
      =     L 0.0;
      A     L 0.0;
      AN    "DOOR_CLEANER_DB".BTM_BRK_HLDR_AUTO_UP_OVR;
      A     "ONE_SECOND_PULSE";
      JNB   M022;
      L     1;
      L     "DOOR_CLEANER_DB".BTM_BRK_HLDR_ATO_UP_DL_T;
      +I;
      T     "DOOR_CLEANER_DB".BTM_BRK_HLDR_ATO_UP_DL_T;
M022: NOP   0;
      A     L 0.0;
      A(;
      L     "DOOR_CLEANER_DB".BTM_BRK_HLDR_ATO_UP_DL_T;
      L     "DOOR_CLEANER_DB".BTM_BRK_HLDR_AUTO_UP_DEL;
      >=I;
      );
      =     "DOOR_CLEANER_DB".BTM_BRK_HLDR_AUTO_UP_OVR;
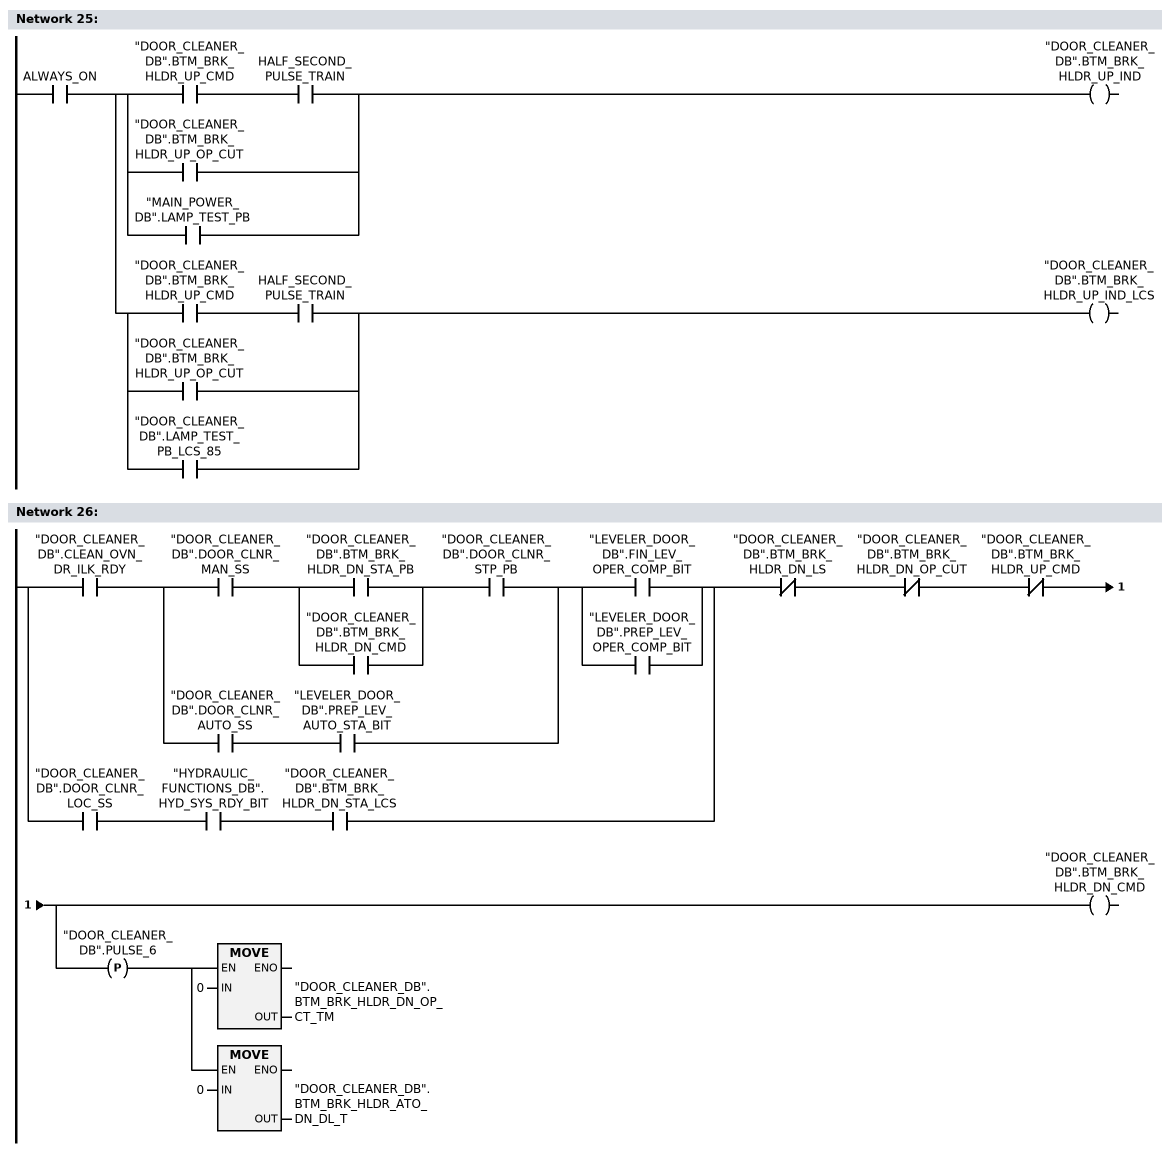
NETWORK
TITLE =
      A     "ALWAYS_ON";
      =     L 0.0;
      A     L 0.0;
      A(;
      A     "DOOR_CLEANER_DB".BTM_BRK_HLDR_UP_CMD;
      A     "HALF_SECOND_PULSE_TRAIN";
      O     "DOOR_CLEANER_DB".BTM_BRK_HLDR_UP_OP_CUT;
      O     "MAIN_POWER_DB".LAMP_TEST_PB;
      );
      =     "DOOR_CLEANER_DB".BTM_BRK_HLDR_UP_IND;
      A     L 0.0;
      A(;
      A     "DOOR_CLEANER_DB".BTM_BRK_HLDR_UP_CMD;
      A     "HALF_SECOND_PULSE_TRAIN";
      O     "DOOR_CLEANER_DB".BTM_BRK_HLDR_UP_OP_CUT;
      O     "DOOR_CLEANER_DB".LAMP_TEST_PB_LCS_85;
      );
      =     "DOOR_CLEANER_DB".BTM_BRK_HLDR_UP_IND_LCS;
NETWORK
TITLE =
      A(;
      A     "DOOR_CLEANER_DB".CLEAN_OVN_DR_ILK_RDY;
      A(;
      A     "DOOR_CLEANER_DB".DOOR_CLNR_MAN_SS;
      A(;
      O     "DOOR_CLEANER_DB".BTM_BRK_HLDR_DN_STA_PB;
      O     "DOOR_CLEANER_DB".BTM_BRK_HLDR_DN_CMD;
      );
      A     "DOOR_CLEANER_DB".DOOR_CLNR_STP_PB;
      O;
      A     "DOOR_CLEANER_DB".DOOR_CLNR_AUTO_SS;
      A     "LEVELER_DOOR_DB".PREP_LEV_AUTO_STA_BIT;
      );
      A(;
      O     "LEVELER_DOOR_DB".FIN_LEV_OPER_COMP_BIT;
      O     "LEVELER_DOOR_DB".PREP_LEV_OPER_COMP_BIT;
      );
      O;
      A     "DOOR_CLEANER_DB".DOOR_CLNR_LOC_SS;
      A     "HYDRAULIC_FUNCTIONS_DB".HYD_SYS_RDY_BIT;
      A     "DOOR_CLEANER_DB".BTM_BRK_HLDR_DN_STA_LCS;
      );
      AN    "DOOR_CLEANER_DB".BTM_BRK_HLDR_DN_LS;
      AN    "DOOR_CLEANER_DB".BTM_BRK_HLDR_DN_OP_CUT;
      AN    "DOOR_CLEANER_DB".BTM_BRK_HLDR_UP_CMD;
      =     L 0.0;
      A     L 0.0;
      BLD   102;
      =     "DOOR_CLEANER_DB".BTM_BRK_HLDR_DN_CMD;
      A     L 0.0;
      FP    "DOOR_CLEANER_DB".PULSE_6;
      =     L 0.1;
      A     L 0.1;
      JNB   M023;
      L     0;
      T     "DOOR_CLEANER_DB".BTM_BRK_HLDR_DN_OP_CT_TM;
M023: NOP   0;
      A     L 0.1;
      JNB   M024;
      L     0;
      T     "DOOR_CLEANER_DB".BTM_BRK_HLDR_ATO_DN_DL_T;
M024: NOP   0;
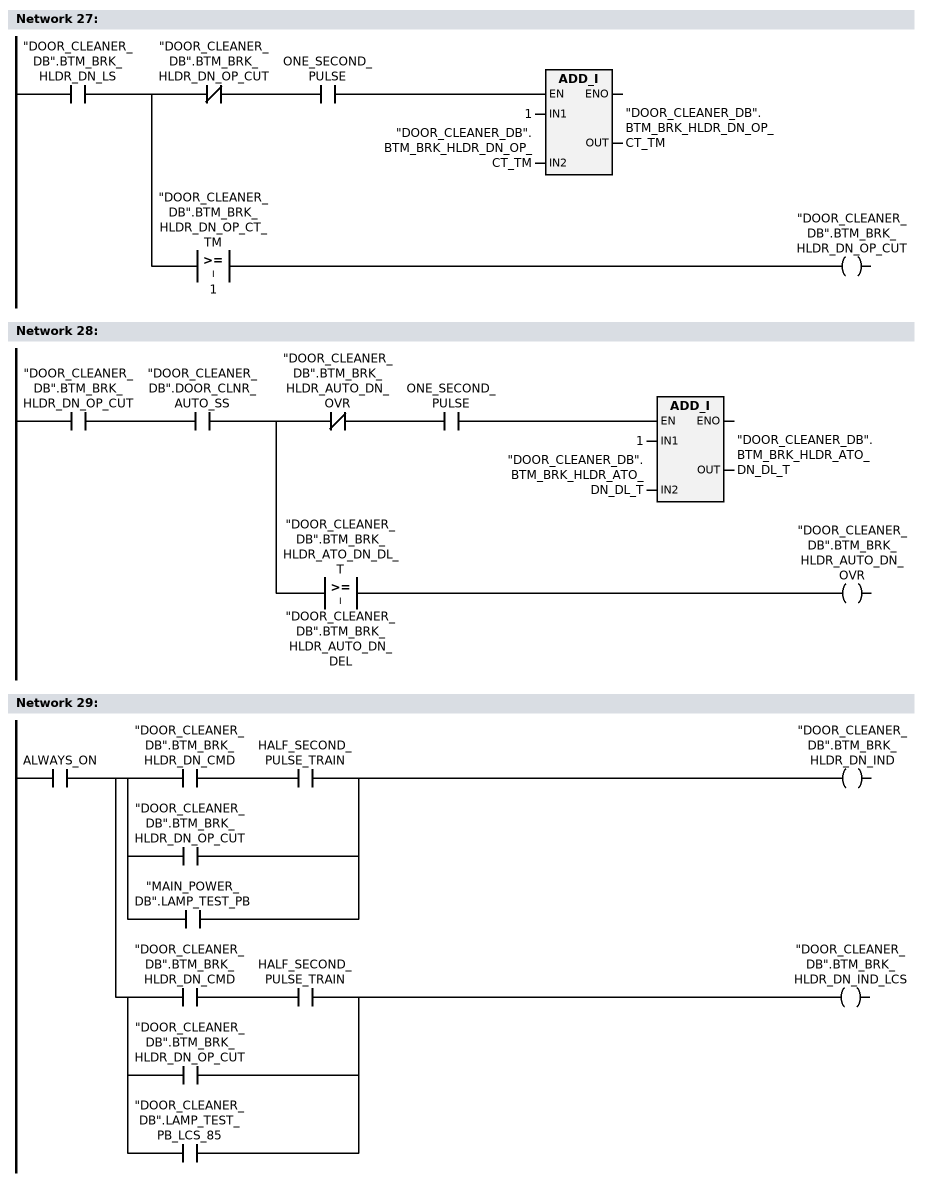
NETWORK
TITLE =
      A     "DOOR_CLEANER_DB".BTM_BRK_HLDR_DN_LS;
      =     L 0.0;
      A     L 0.0;
      AN    "DOOR_CLEANER_DB".BTM_BRK_HLDR_DN_OP_CUT;
      A     "ONE_SECOND_PULSE";
      JNB   M025;
      L     1;
      L     "DOOR_CLEANER_DB".BTM_BRK_HLDR_DN_OP_CT_TM;
      +I;
      T     "DOOR_CLEANER_DB".BTM_BRK_HLDR_DN_OP_CT_TM;
M025: NOP   0;
      A     L 0.0;
      A(;
      L     "DOOR_CLEANER_DB".BTM_BRK_HLDR_DN_OP_CT_TM;
      L     1;
      >=I;
      );
      =     "DOOR_CLEANER_DB".BTM_BRK_HLDR_DN_OP_CUT;
NETWORK
TITLE =
      A     "DOOR_CLEANER_DB".BTM_BRK_HLDR_DN_OP_CUT;
      A     "DOOR_CLEANER_DB".DOOR_CLNR_AUTO_SS;
      =     L 0.0;
      A     L 0.0;
      AN    "DOOR_CLEANER_DB".BTM_BRK_HLDR_AUTO_DN_OVR;
      A     "ONE_SECOND_PULSE";
      JNB   M026;
      L     1;
      L     "DOOR_CLEANER_DB".BTM_BRK_HLDR_ATO_DN_DL_T;
      +I;
      T     "DOOR_CLEANER_DB".BTM_BRK_HLDR_ATO_DN_DL_T;
M026: NOP   0;
      A     L 0.0;
      A(;
      L     "DOOR_CLEANER_DB".BTM_BRK_HLDR_ATO_DN_DL_T;
      L     "DOOR_CLEANER_DB".BTM_BRK_HLDR_AUTO_DN_DEL;
      >=I;
      );
      =     "DOOR_CLEANER_DB".BTM_BRK_HLDR_AUTO_DN_OVR;
NETWORK
TITLE =
      A     "ALWAYS_ON";
      =     L 0.0;
      A     L 0.0;
      A(;
      A     "DOOR_CLEANER_DB".BTM_BRK_HLDR_DN_CMD;
      A     "HALF_SECOND_PULSE_TRAIN";
      O     "DOOR_CLEANER_DB".BTM_BRK_HLDR_DN_OP_CUT;
      O     "MAIN_POWER_DB".LAMP_TEST_PB;
      );
      =     "DOOR_CLEANER_DB".BTM_BRK_HLDR_DN_IND;
      A     L 0.0;
      A(;
      A     "DOOR_CLEANER_DB".BTM_BRK_HLDR_DN_CMD;
      A     "HALF_SECOND_PULSE_TRAIN";
      O     "DOOR_CLEANER_DB".BTM_BRK_HLDR_DN_OP_CUT;
      O     "DOOR_CLEANER_DB".LAMP_TEST_PB_LCS_85;
      );
      =     "DOOR_CLEANER_DB".BTM_BRK_HLDR_DN_IND_LCS;
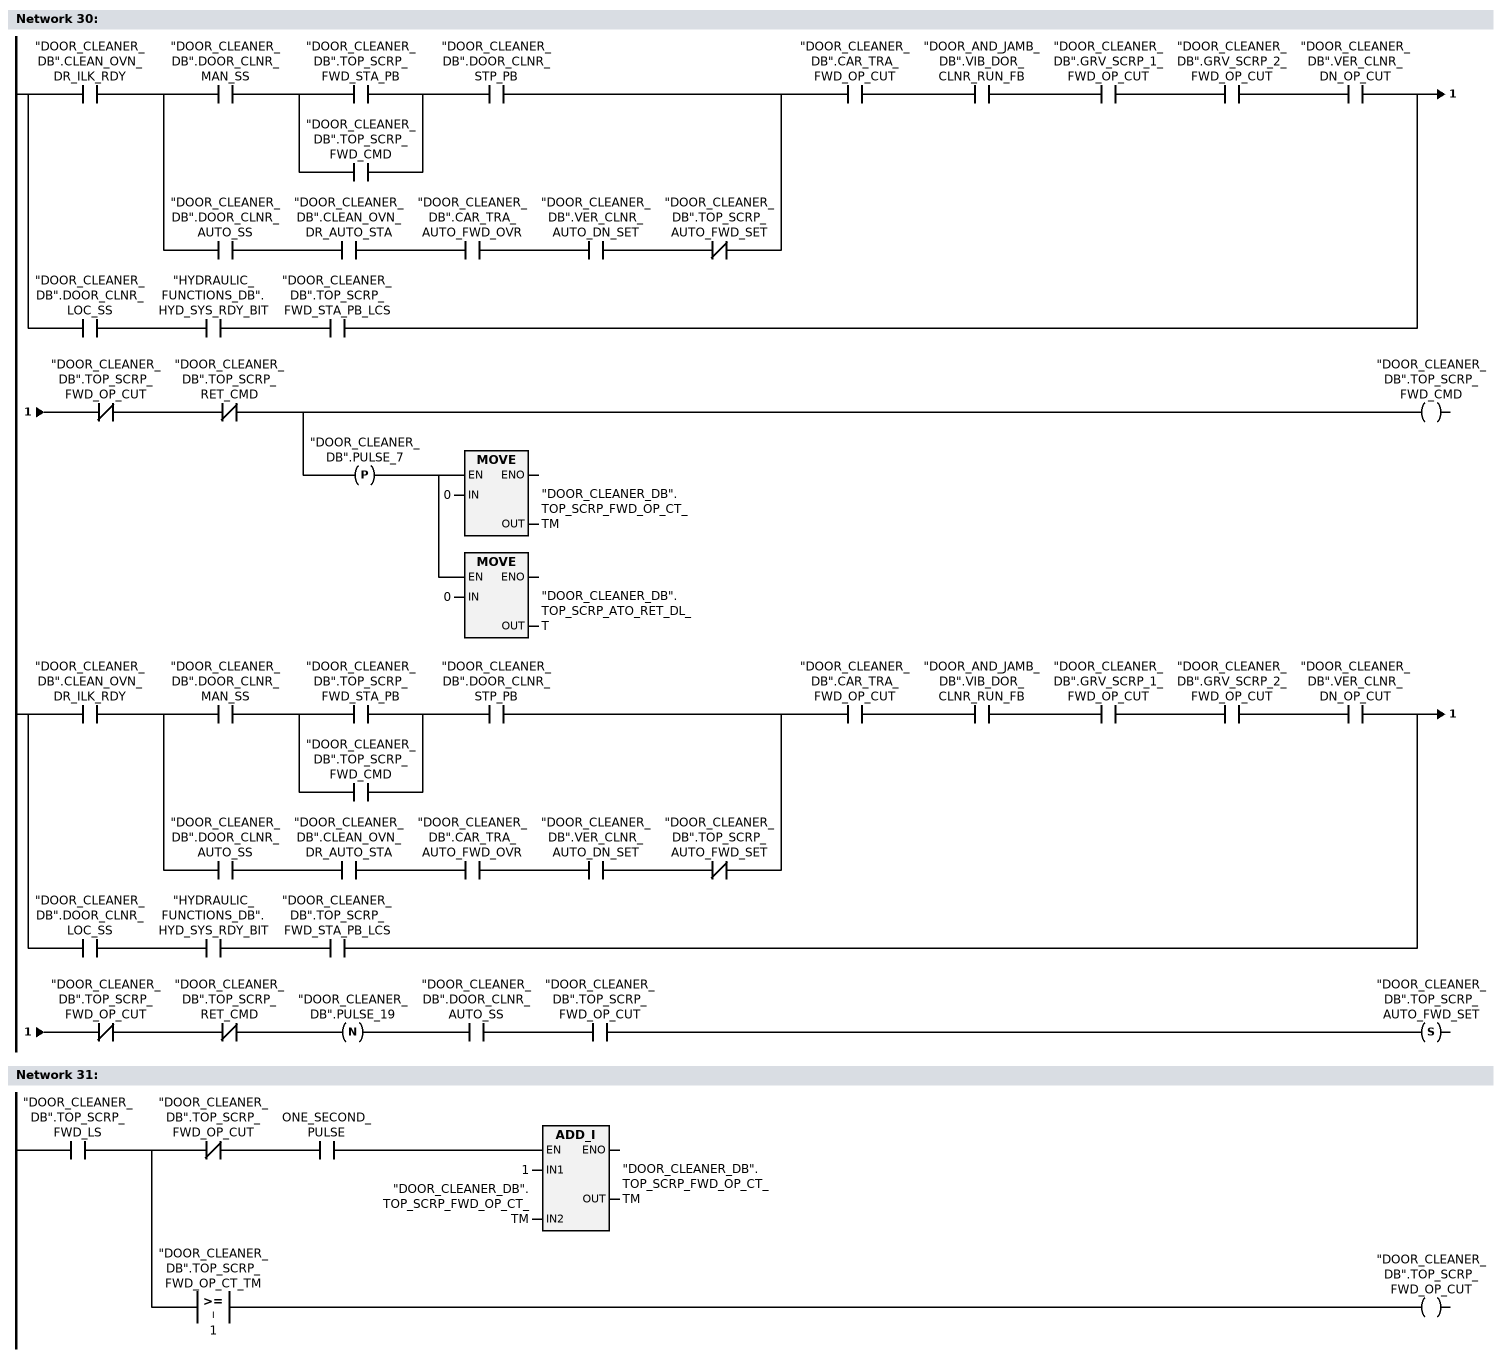
NETWORK
TITLE =
      A(;
      A     "DOOR_CLEANER_DB".CLEAN_OVN_DR_ILK_RDY;
      A(;
      A     "DOOR_CLEANER_DB".DOOR_CLNR_MAN_SS;
      A(;
      O     "DOOR_CLEANER_DB".TOP_SCRP_FWD_STA_PB;
      O     "DOOR_CLEANER_DB".TOP_SCRP_FWD_CMD;
      );
      A     "DOOR_CLEANER_DB".DOOR_CLNR_STP_PB;
      O;
      A     "DOOR_CLEANER_DB".DOOR_CLNR_AUTO_SS;
      A     "DOOR_CLEANER_DB".CLEAN_OVN_DR_AUTO_STA;
      A     "DOOR_CLEANER_DB".CAR_TRA_AUTO_FWD_OVR;
      A     "DOOR_CLEANER_DB".VER_CLNR_AUTO_DN_SET;
      AN    "DOOR_CLEANER_DB".TOP_SCRP_AUTO_FWD_SET;
      );
      A     "DOOR_CLEANER_DB".CAR_TRA_FWD_OP_CUT;
      A     "DOOR_AND_JAMB_DB".VIB_DOR_CLNR_RUN_FB;
      A     "DOOR_CLEANER_DB".GRV_SCRP_1_FWD_OP_CUT;
      A     "DOOR_CLEANER_DB".GRV_SCRP_2_FWD_OP_CUT;
      A     "DOOR_CLEANER_DB".VER_CLNR_DN_OP_CUT;
      O;
      A     "DOOR_CLEANER_DB".DOOR_CLNR_LOC_SS;
      A     "HYDRAULIC_FUNCTIONS_DB".HYD_SYS_RDY_BIT;
      A     "DOOR_CLEANER_DB".TOP_SCRP_FWD_STA_PB_LCS;
      );
      AN    "DOOR_CLEANER_DB".TOP_SCRP_FWD_OP_CUT;
      AN    "DOOR_CLEANER_DB".TOP_SCRP_RET_CMD;
      =     L 0.0;
      A     L 0.0;
      BLD   102;
      =     "DOOR_CLEANER_DB".TOP_SCRP_FWD_CMD;
      A(;
      A     L 0.0;
      FN    "DOOR_CLEANER_DB".PULSE_19;
      );
      A     "DOOR_CLEANER_DB".DOOR_CLNR_AUTO_SS;
      A     "DOOR_CLEANER_DB".TOP_SCRP_FWD_OP_CUT;
      S     "DOOR_CLEANER_DB".TOP_SCRP_AUTO_FWD_SET;
      A     L 0.0;
      FP    "DOOR_CLEANER_DB".PULSE_7;
      =     L 0.1;
      A     L 0.1;
      JNB   M027;
      L     0;
      T     "DOOR_CLEANER_DB".TOP_SCRP_FWD_OP_CT_TM;
M027: NOP   0;
      A     L 0.1;
      JNB   M028;
      L     0;
      T     "DOOR_CLEANER_DB".TOP_SCRP_ATO_RET_DL_T;
M028: NOP   0;
NETWORK
TITLE =
      A     "DOOR_CLEANER_DB".TOP_SCRP_FWD_LS;
      =     L 0.0;
      A     L 0.0;
      AN    "DOOR_CLEANER_DB".TOP_SCRP_FWD_OP_CUT;
      A     "ONE_SECOND_PULSE";
      JNB   M029;
      L     1;
      L     "DOOR_CLEANER_DB".TOP_SCRP_FWD_OP_CT_TM;
      +I;
      T     "DOOR_CLEANER_DB".TOP_SCRP_FWD_OP_CT_TM;
M029: NOP   0;
      A     L 0.0;
      A(;
      L     "DOOR_CLEANER_DB".TOP_SCRP_FWD_OP_CT_TM;
      L     1;
      >=I;
      );
      =     "DOOR_CLEANER_DB".TOP_SCRP_FWD_OP_CUT;
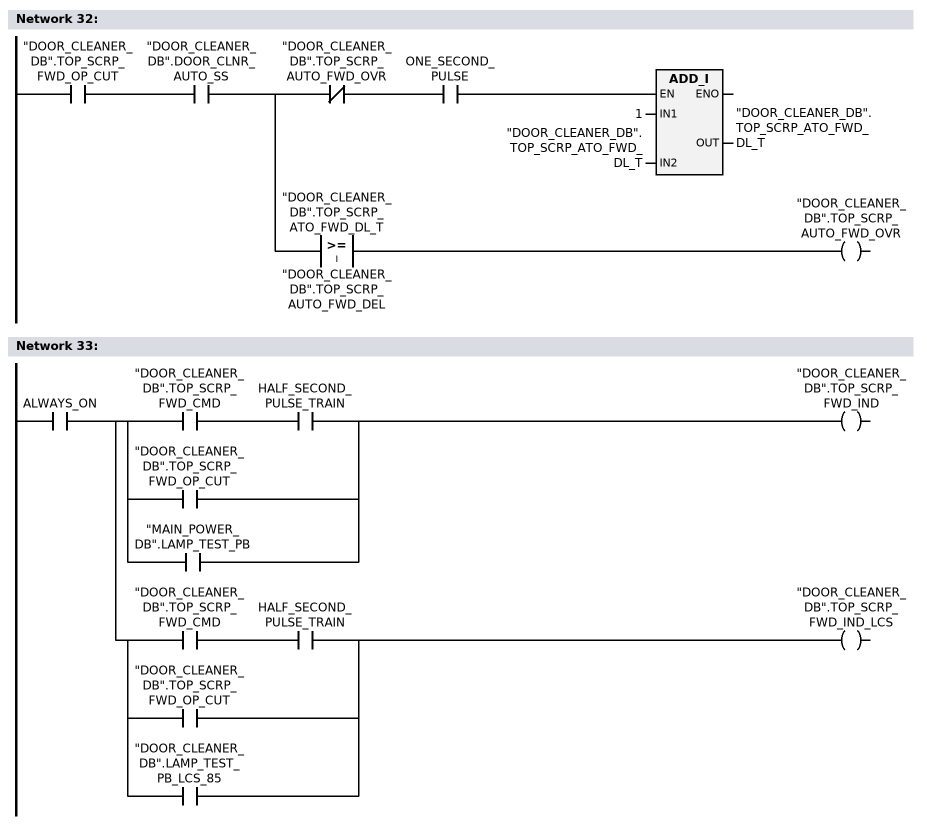
NETWORK
TITLE =
      A     "DOOR_CLEANER_DB".TOP_SCRP_FWD_OP_CUT;
      A     "DOOR_CLEANER_DB".DOOR_CLNR_AUTO_SS;
      =     L 0.0;
      A     L 0.0;
      AN    "DOOR_CLEANER_DB".TOP_SCRP_AUTO_FWD_OVR;
      A     "ONE_SECOND_PULSE";
      JNB   M030;
      L     1;
      L     "DOOR_CLEANER_DB".TOP_SCRP_ATO_FWD_DL_T;
      +I;
      T     "DOOR_CLEANER_DB".TOP_SCRP_ATO_FWD_DL_T;
M030: NOP   0;
      A     L 0.0;
      A(;
      L     "DOOR_CLEANER_DB".TOP_SCRP_ATO_FWD_DL_T;
      L     "DOOR_CLEANER_DB".TOP_SCRP_AUTO_FWD_DEL;
      >=I;
      );
      =     "DOOR_CLEANER_DB".TOP_SCRP_AUTO_FWD_OVR;
NETWORK
TITLE =
      A     "ALWAYS_ON";
      =     L 0.0;
      A     L 0.0;
      A(;
      A     "DOOR_CLEANER_DB".TOP_SCRP_FWD_CMD;
      A     "HALF_SECOND_PULSE_TRAIN";
      O     "DOOR_CLEANER_DB".TOP_SCRP_FWD_OP_CUT;
      O     "MAIN_POWER_DB".LAMP_TEST_PB;
      );
      =     "DOOR_CLEANER_DB".TOP_SCRP_FWD_IND;
      A     L 0.0;
      A(;
      A     "DOOR_CLEANER_DB".TOP_SCRP_FWD_CMD;
      A     "HALF_SECOND_PULSE_TRAIN";
      O     "DOOR_CLEANER_DB".TOP_SCRP_FWD_OP_CUT;
      O     "DOOR_CLEANER_DB".LAMP_TEST_PB_LCS_85;
      );
      =     "DOOR_CLEANER_DB".TOP_SCRP_FWD_IND_LCS;
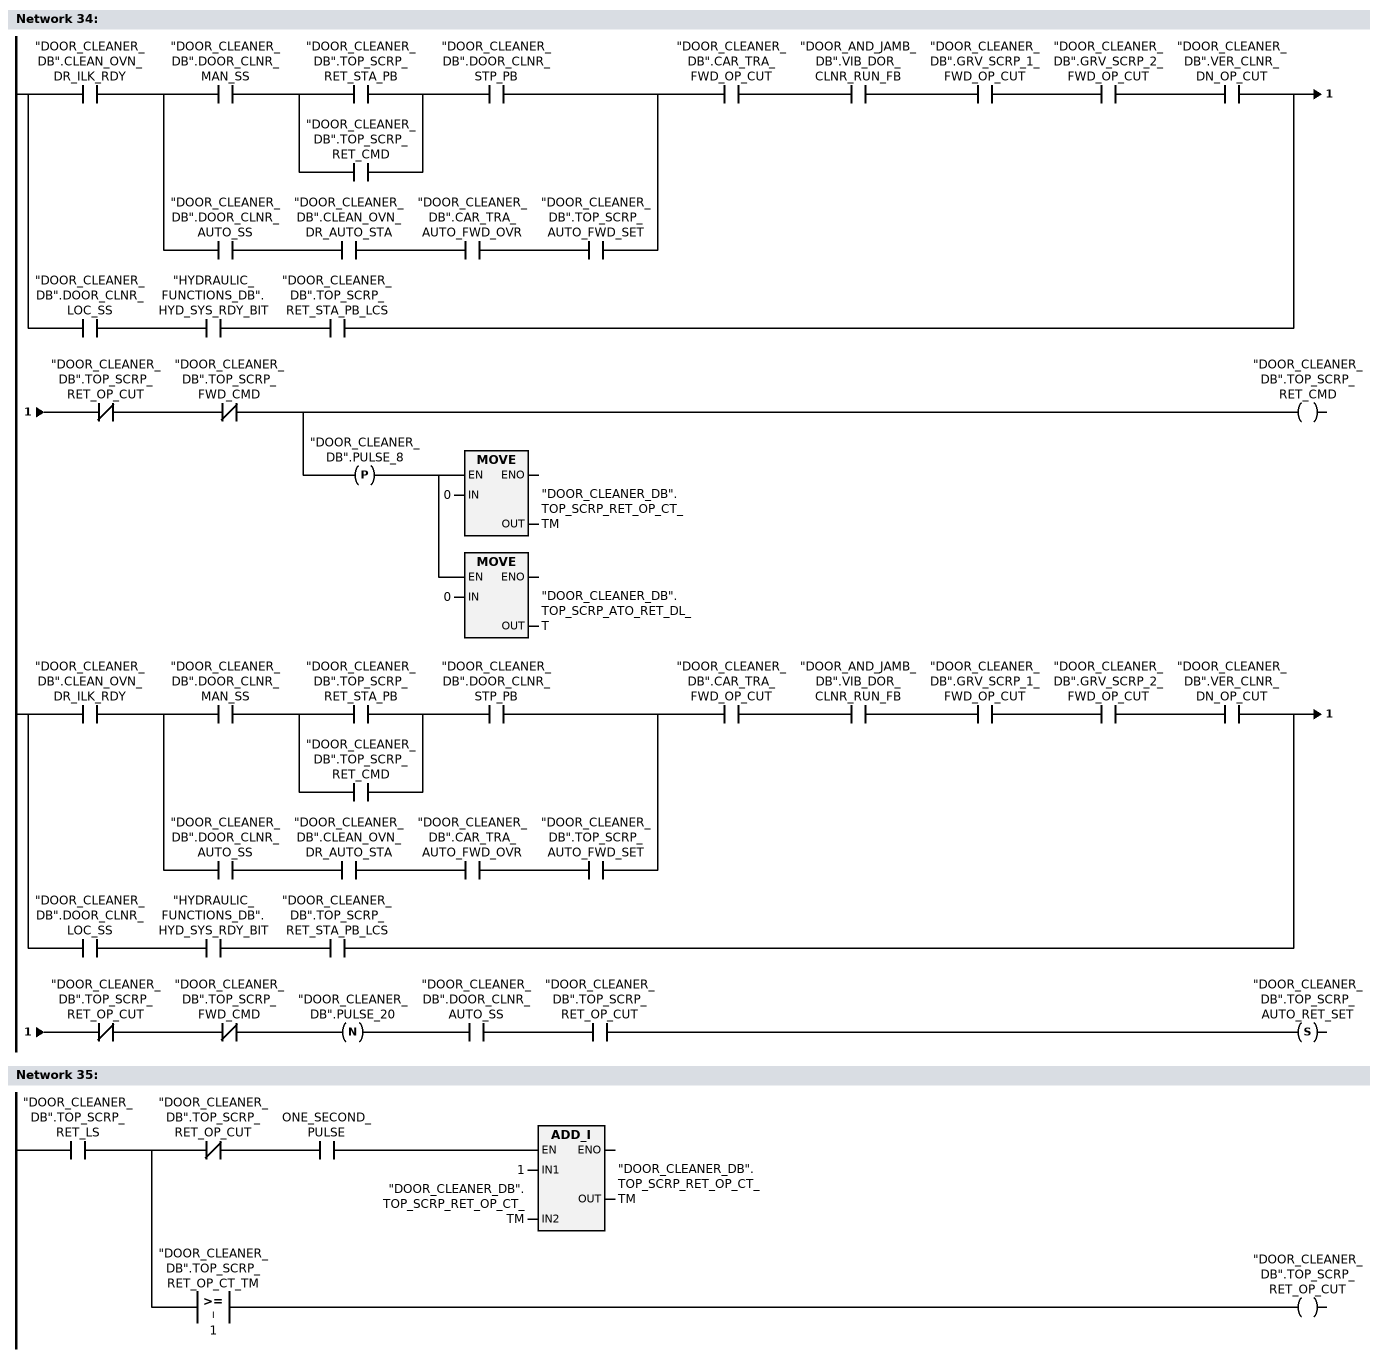
NETWORK
TITLE =
      A(;
      A     "DOOR_CLEANER_DB".CLEAN_OVN_DR_ILK_RDY;
      A(;
      A     "DOOR_CLEANER_DB".DOOR_CLNR_MAN_SS;
      A(;
      O     "DOOR_CLEANER_DB".TOP_SCRP_RET_STA_PB;
      O     "DOOR_CLEANER_DB".TOP_SCRP_RET_CMD;
      );
      A     "DOOR_CLEANER_DB".DOOR_CLNR_STP_PB;
      O;
      A     "DOOR_CLEANER_DB".DOOR_CLNR_AUTO_SS;
      A     "DOOR_CLEANER_DB".CLEAN_OVN_DR_AUTO_STA;
      A     "DOOR_CLEANER_DB".CAR_TRA_AUTO_FWD_OVR;
      A     "DOOR_CLEANER_DB".TOP_SCRP_AUTO_FWD_SET;
      );
      A     "DOOR_CLEANER_DB".CAR_TRA_FWD_OP_CUT;
      A     "DOOR_AND_JAMB_DB".VIB_DOR_CLNR_RUN_FB;
      A     "DOOR_CLEANER_DB".GRV_SCRP_1_FWD_OP_CUT;
      A     "DOOR_CLEANER_DB".GRV_SCRP_2_FWD_OP_CUT;
      A     "DOOR_CLEANER_DB".VER_CLNR_DN_OP_CUT;
      O;
      A     "DOOR_CLEANER_DB".DOOR_CLNR_LOC_SS;
      A     "HYDRAULIC_FUNCTIONS_DB".HYD_SYS_RDY_BIT;
      A     "DOOR_CLEANER_DB".TOP_SCRP_RET_STA_PB_LCS;
      );
      AN    "DOOR_CLEANER_DB".TOP_SCRP_RET_OP_CUT;
      AN    "DOOR_CLEANER_DB".TOP_SCRP_FWD_CMD;
      =     L 0.0;
      A     L 0.0;
      BLD   102;
      =     "DOOR_CLEANER_DB".TOP_SCRP_RET_CMD;
      A(;
      A     L 0.0;
      FN    "DOOR_CLEANER_DB".PULSE_20;
      );
      A     "DOOR_CLEANER_DB".DOOR_CLNR_AUTO_SS;
      A     "DOOR_CLEANER_DB".TOP_SCRP_RET_OP_CUT;
      S     "DOOR_CLEANER_DB".TOP_SCRP_AUTO_RET_SET;
      A     L 0.0;
      FP    "DOOR_CLEANER_DB".PULSE_8;
      =     L 0.1;
      A     L 0.1;
      JNB   M031;
      L     0;
      T     "DOOR_CLEANER_DB".TOP_SCRP_RET_OP_CT_TM;
M031: NOP   0;
      A     L 0.1;
      JNB   M032;
      L     0;
      T     "DOOR_CLEANER_DB".TOP_SCRP_ATO_RET_DL_T;
M032: NOP   0;
NETWORK
TITLE =
      A     "DOOR_CLEANER_DB".TOP_SCRP_RET_LS;
      =     L 0.0;
      A     L 0.0;
      AN    "DOOR_CLEANER_DB".TOP_SCRP_RET_OP_CUT;
      A     "ONE_SECOND_PULSE";
      JNB   M033;
      L     1;
      L     "DOOR_CLEANER_DB".TOP_SCRP_RET_OP_CT_TM;
      +I;
      T     "DOOR_CLEANER_DB".TOP_SCRP_RET_OP_CT_TM;
M033: NOP   0;
      A     L 0.0;
      A(;
      L     "DOOR_CLEANER_DB".TOP_SCRP_RET_OP_CT_TM;
      L     1;
      >=I;
      );
      =     "DOOR_CLEANER_DB".TOP_SCRP_RET_OP_CUT;
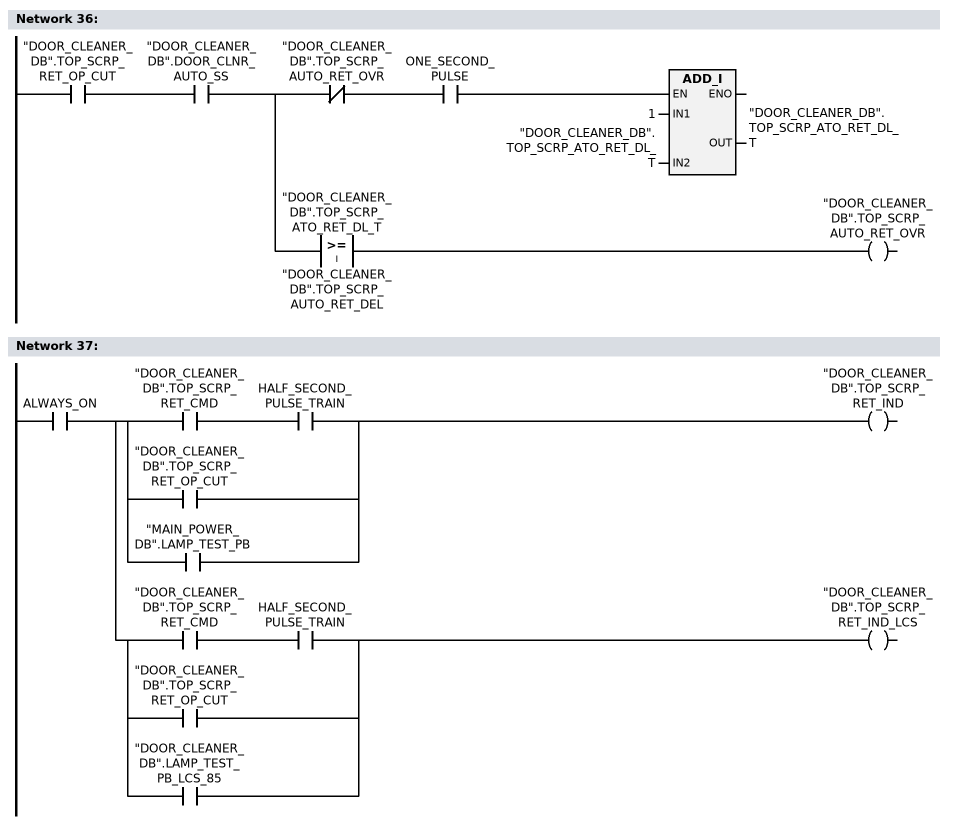
NETWORK
TITLE =
      A     "DOOR_CLEANER_DB".TOP_SCRP_RET_OP_CUT;
      A     "DOOR_CLEANER_DB".DOOR_CLNR_AUTO_SS;
      =     L 0.0;
      A     L 0.0;
      AN    "DOOR_CLEANER_DB".TOP_SCRP_AUTO_RET_OVR;
      A     "ONE_SECOND_PULSE";
      JNB   M034;
      L     1;
      L     "DOOR_CLEANER_DB".TOP_SCRP_ATO_RET_DL_T;
      +I;
      T     "DOOR_CLEANER_DB".TOP_SCRP_ATO_RET_DL_T;
M034: NOP   0;
      A     L 0.0;
      A(;
      L     "DOOR_CLEANER_DB".TOP_SCRP_ATO_RET_DL_T;
      L     "DOOR_CLEANER_DB".TOP_SCRP_AUTO_RET_DEL;
      >=I;
      );
      =     "DOOR_CLEANER_DB".TOP_SCRP_AUTO_RET_OVR;
NETWORK
TITLE =
      A     "ALWAYS_ON";
      =     L 0.0;
      A     L 0.0;
      A(;
      A     "DOOR_CLEANER_DB".TOP_SCRP_RET_CMD;
      A     "HALF_SECOND_PULSE_TRAIN";
      O     "DOOR_CLEANER_DB".TOP_SCRP_RET_OP_CUT;
      O     "MAIN_POWER_DB".LAMP_TEST_PB;
      );
      =     "DOOR_CLEANER_DB".TOP_SCRP_RET_IND;
      A     L 0.0;
      A(;
      A     "DOOR_CLEANER_DB".TOP_SCRP_RET_CMD;
      A     "HALF_SECOND_PULSE_TRAIN";
      O     "DOOR_CLEANER_DB".TOP_SCRP_RET_OP_CUT;
      O     "DOOR_CLEANER_DB".LAMP_TEST_PB_LCS_85;
      );
      =     "DOOR_CLEANER_DB".TOP_SCRP_RET_IND_LCS;
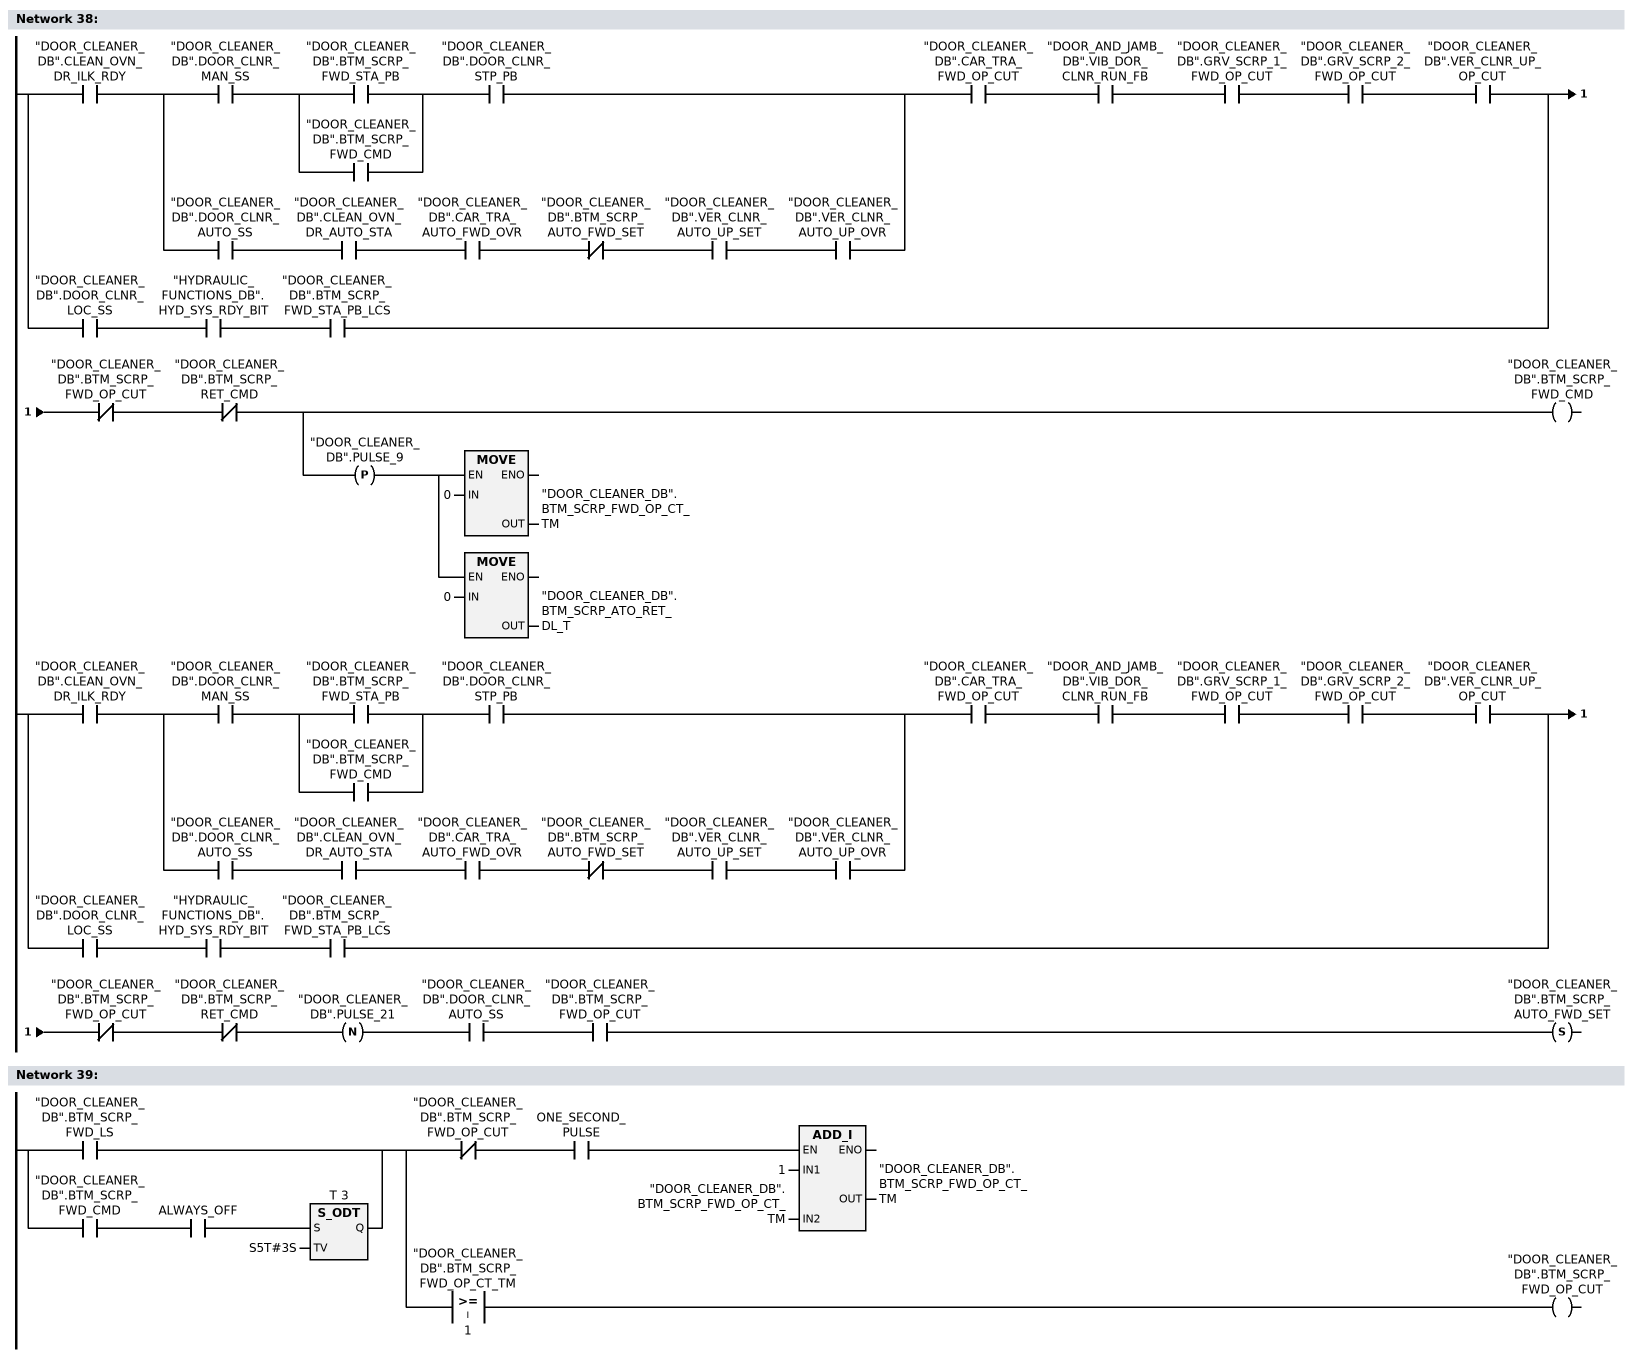
NETWORK
TITLE =
      A(;
      A     "DOOR_CLEANER_DB".CLEAN_OVN_DR_ILK_RDY;
      A(;
      A     "DOOR_CLEANER_DB".DOOR_CLNR_MAN_SS;
      A(;
      O     "DOOR_CLEANER_DB".BTM_SCRP_FWD_STA_PB;
      O     "DOOR_CLEANER_DB".BTM_SCRP_FWD_CMD;
      );
      A     "DOOR_CLEANER_DB".DOOR_CLNR_STP_PB;
      O;
      A     "DOOR_CLEANER_DB".DOOR_CLNR_AUTO_SS;
      A     "DOOR_CLEANER_DB".CLEAN_OVN_DR_AUTO_STA;
      A     "DOOR_CLEANER_DB".CAR_TRA_AUTO_FWD_OVR;
      AN    "DOOR_CLEANER_DB".BTM_SCRP_AUTO_FWD_SET;
      A     "DOOR_CLEANER_DB".VER_CLNR_AUTO_UP_SET;
      A     "DOOR_CLEANER_DB".VER_CLNR_AUTO_UP_OVR;
      );
      A     "DOOR_CLEANER_DB".CAR_TRA_FWD_OP_CUT;
      A     "DOOR_AND_JAMB_DB".VIB_DOR_CLNR_RUN_FB;
      A     "DOOR_CLEANER_DB".GRV_SCRP_1_FWD_OP_CUT;
      A     "DOOR_CLEANER_DB".GRV_SCRP_2_FWD_OP_CUT;
      A     "DOOR_CLEANER_DB".VER_CLNR_UP_OP_CUT;
      O;
      A     "DOOR_CLEANER_DB".DOOR_CLNR_LOC_SS;
      A     "HYDRAULIC_FUNCTIONS_DB".HYD_SYS_RDY_BIT;
      A     "DOOR_CLEANER_DB".BTM_SCRP_FWD_STA_PB_LCS;
      );
      AN    "DOOR_CLEANER_DB".BTM_SCRP_FWD_OP_CUT;
      AN    "DOOR_CLEANER_DB".BTM_SCRP_RET_CMD;
      =     L 0.0;
      A     L 0.0;
      BLD   102;
      =     "DOOR_CLEANER_DB".BTM_SCRP_FWD_CMD;
      A(;
      A     L 0.0;
      FN    "DOOR_CLEANER_DB".PULSE_21;
      );
      A     "DOOR_CLEANER_DB".DOOR_CLNR_AUTO_SS;
      A     "DOOR_CLEANER_DB".BTM_SCRP_FWD_OP_CUT;
      S     "DOOR_CLEANER_DB".BTM_SCRP_AUTO_FWD_SET;
      A     L 0.0;
      FP    "DOOR_CLEANER_DB".PULSE_9;
      =     L 0.1;
      A     L 0.1;
      JNB   M035;
      L     0;
      T     "DOOR_CLEANER_DB".BTM_SCRP_FWD_OP_CT_TM;
M035: NOP   0;
      A     L 0.1;
      JNB   M036;
      L     0;
      T     "DOOR_CLEANER_DB".BTM_SCRP_ATO_RET_DL_T;
M036: NOP   0;
NETWORK
TITLE =
      O     "DOOR_CLEANER_DB".BTM_SCRP_FWD_LS;
      O(;
      A     "DOOR_CLEANER_DB".BTM_SCRP_FWD_CMD;
      A     "ALWAYS_OFF";
      L     S5T#3S;
      SD    T 3;
      NOP   0;
      NOP   0;
      NOP   0;
      A     T 3;
      );
      =     L 0.0;
      A     L 0.0;
      AN    "DOOR_CLEANER_DB".BTM_SCRP_FWD_OP_CUT;
      A     "ONE_SECOND_PULSE";
      JNB   M037;
      L     1;
      L     "DOOR_CLEANER_DB".BTM_SCRP_FWD_OP_CT_TM;
      +I;
      T     "DOOR_CLEANER_DB".BTM_SCRP_FWD_OP_CT_TM;
M037: NOP   0;
      A     L 0.0;
      A(;
      L     "DOOR_CLEANER_DB".BTM_SCRP_FWD_OP_CT_TM;
      L     1;
      >=I;
      );
      =     "DOOR_CLEANER_DB".BTM_SCRP_FWD_OP_CUT;
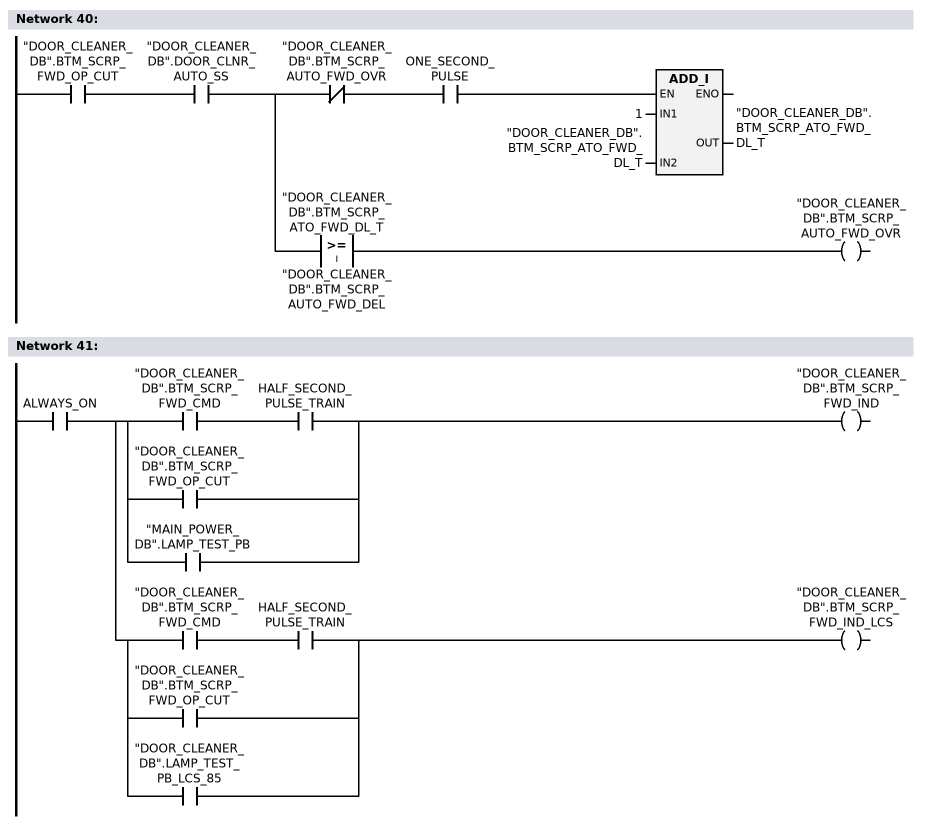
NETWORK
TITLE =
      A     "DOOR_CLEANER_DB".BTM_SCRP_FWD_OP_CUT;
      A     "DOOR_CLEANER_DB".DOOR_CLNR_AUTO_SS;
      =     L 0.0;
      A     L 0.0;
      AN    "DOOR_CLEANER_DB".BTM_SCRP_AUTO_FWD_OVR;
      A     "ONE_SECOND_PULSE";
      JNB   M038;
      L     1;
      L     "DOOR_CLEANER_DB".BTM_SCRP_ATO_FWD_DL_T;
      +I;
      T     "DOOR_CLEANER_DB".BTM_SCRP_ATO_FWD_DL_T;
M038: NOP   0;
      A     L 0.0;
      A(;
      L     "DOOR_CLEANER_DB".BTM_SCRP_ATO_FWD_DL_T;
      L     "DOOR_CLEANER_DB".BTM_SCRP_AUTO_FWD_DEL;
      >=I;
      );
      =     "DOOR_CLEANER_DB".BTM_SCRP_AUTO_FWD_OVR;
NETWORK
TITLE =
      A     "ALWAYS_ON";
      =     L 0.0;
      A     L 0.0;
      A(;
      A     "DOOR_CLEANER_DB".BTM_SCRP_FWD_CMD;
      A     "HALF_SECOND_PULSE_TRAIN";
      O     "DOOR_CLEANER_DB".BTM_SCRP_FWD_OP_CUT;
      O     "MAIN_POWER_DB".LAMP_TEST_PB;
      );
      =     "DOOR_CLEANER_DB".BTM_SCRP_FWD_IND;
      A     L 0.0;
      A(;
      A     "DOOR_CLEANER_DB".BTM_SCRP_FWD_CMD;
      A     "HALF_SECOND_PULSE_TRAIN";
      O     "DOOR_CLEANER_DB".BTM_SCRP_FWD_OP_CUT;
      O     "DOOR_CLEANER_DB".LAMP_TEST_PB_LCS_85;
      );
      =     "DOOR_CLEANER_DB".BTM_SCRP_FWD_IND_LCS;
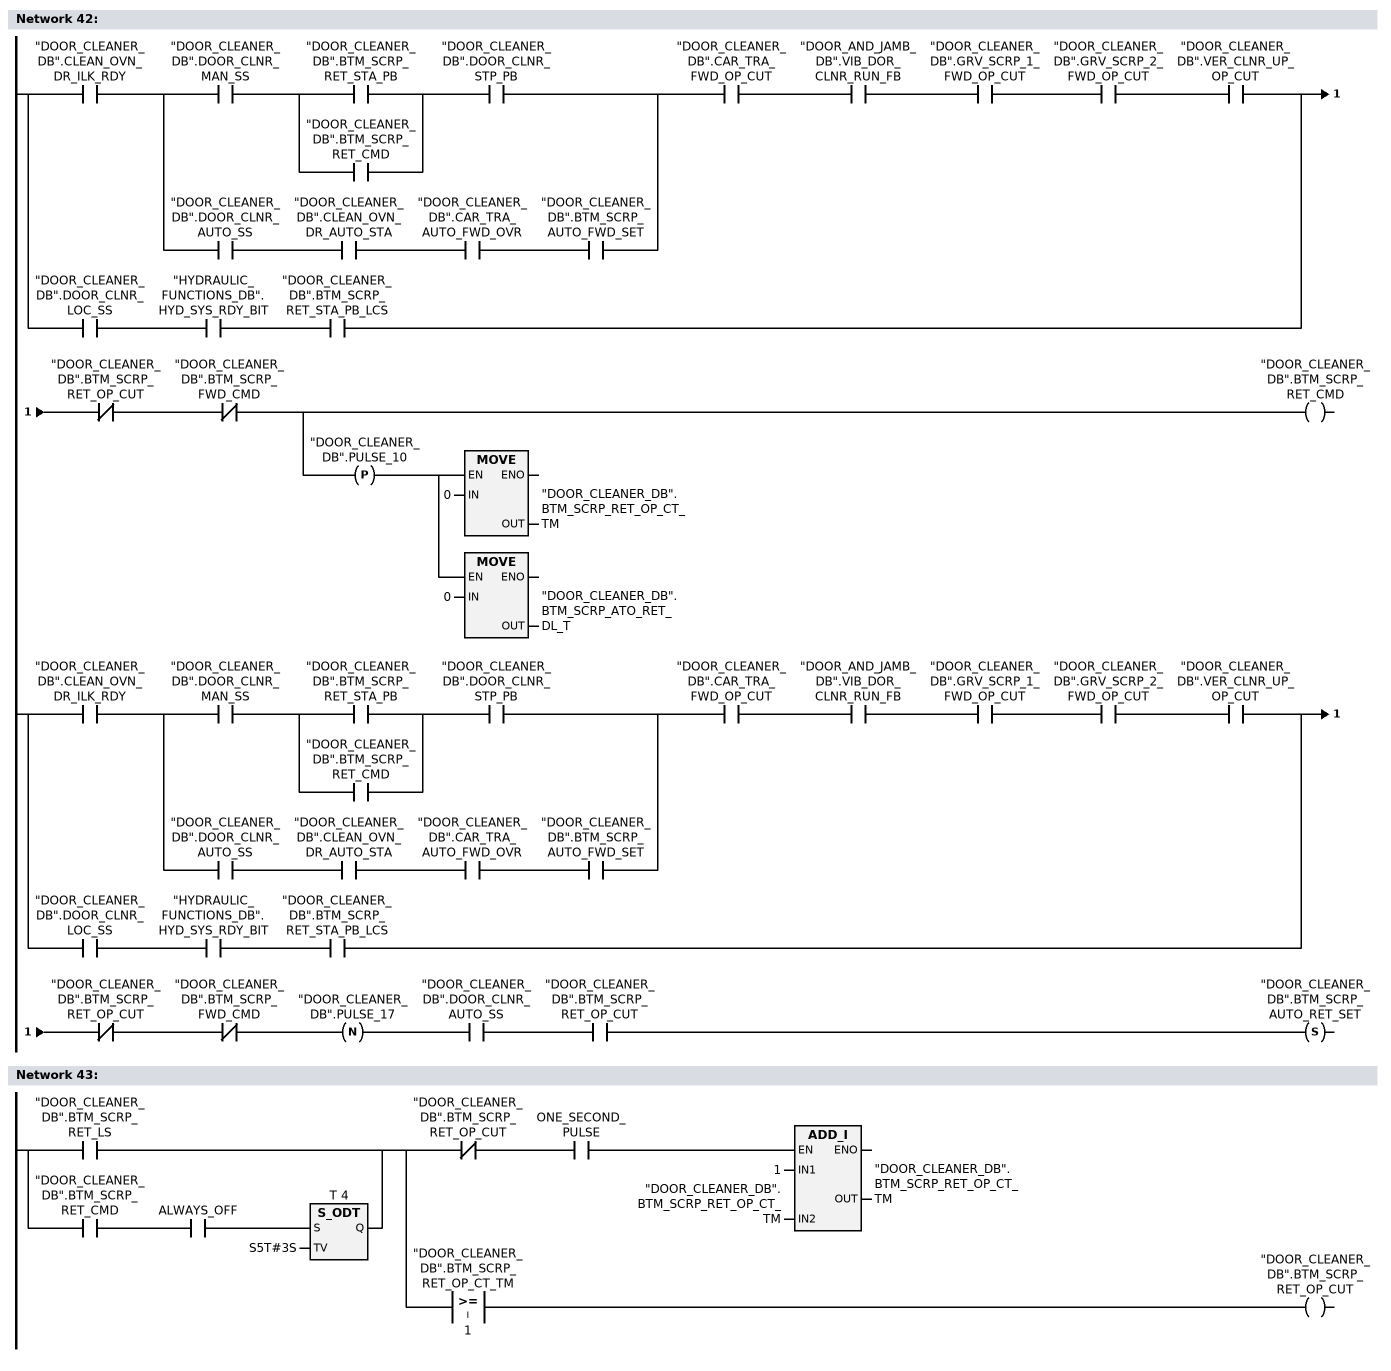
NETWORK
TITLE =
      A(;
      A     "DOOR_CLEANER_DB".CLEAN_OVN_DR_ILK_RDY;
      A(;
      A     "DOOR_CLEANER_DB".DOOR_CLNR_MAN_SS;
      A(;
      O     "DOOR_CLEANER_DB".BTM_SCRP_RET_STA_PB;
      O     "DOOR_CLEANER_DB".BTM_SCRP_RET_CMD;
      );
      A     "DOOR_CLEANER_DB".DOOR_CLNR_STP_PB;
      O;
      A     "DOOR_CLEANER_DB".DOOR_CLNR_AUTO_SS;
      A     "DOOR_CLEANER_DB".CLEAN_OVN_DR_AUTO_STA;
      A     "DOOR_CLEANER_DB".CAR_TRA_AUTO_FWD_OVR;
      A     "DOOR_CLEANER_DB".BTM_SCRP_AUTO_FWD_SET;
      );
      A     "DOOR_CLEANER_DB".CAR_TRA_FWD_OP_CUT;
      A     "DOOR_AND_JAMB_DB".VIB_DOR_CLNR_RUN_FB;
      A     "DOOR_CLEANER_DB".GRV_SCRP_1_FWD_OP_CUT;
      A     "DOOR_CLEANER_DB".GRV_SCRP_2_FWD_OP_CUT;
      A     "DOOR_CLEANER_DB".VER_CLNR_UP_OP_CUT;
      O;
      A     "DOOR_CLEANER_DB".DOOR_CLNR_LOC_SS;
      A     "HYDRAULIC_FUNCTIONS_DB".HYD_SYS_RDY_BIT;
      A     "DOOR_CLEANER_DB".BTM_SCRP_RET_STA_PB_LCS;
      );
      AN    "DOOR_CLEANER_DB".BTM_SCRP_RET_OP_CUT;
      AN    "DOOR_CLEANER_DB".BTM_SCRP_FWD_CMD;
      =     L 0.0;
      A     L 0.0;
      BLD   102;
      =     "DOOR_CLEANER_DB".BTM_SCRP_RET_CMD;
      A(;
      A     L 0.0;
      FN    "DOOR_CLEANER_DB".PULSE_17;
      );
      A     "DOOR_CLEANER_DB".DOOR_CLNR_AUTO_SS;
      A     "DOOR_CLEANER_DB".BTM_SCRP_RET_OP_CUT;
      S     "DOOR_CLEANER_DB".BTM_SCRP_AUTO_RET_SET;
      A     L 0.0;
      FP    "DOOR_CLEANER_DB".PULSE_10;
      =     L 0.1;
      A     L 0.1;
      JNB   M039;
      L     0;
      T     "DOOR_CLEANER_DB".BTM_SCRP_RET_OP_CT_TM;
M039: NOP   0;
      A     L 0.1;
      JNB   M040;
      L     0;
      T     "DOOR_CLEANER_DB".BTM_SCRP_ATO_RET_DL_T;
M040: NOP   0;
NETWORK
TITLE =
      O     "DOOR_CLEANER_DB".BTM_SCRP_RET_LS;
      O(;
      A     "DOOR_CLEANER_DB".BTM_SCRP_RET_CMD;
      A     "ALWAYS_OFF";
      L     S5T#3S;
      SD    T 4;
      NOP   0;
      NOP   0;
      NOP   0;
      A     T 4;
      );
      =     L 0.0;
      A     L 0.0;
      AN    "DOOR_CLEANER_DB".BTM_SCRP_RET_OP_CUT;
      A     "ONE_SECOND_PULSE";
      JNB   M041;
      L     1;
      L     "DOOR_CLEANER_DB".BTM_SCRP_RET_OP_CT_TM;
      +I;
      T     "DOOR_CLEANER_DB".BTM_SCRP_RET_OP_CT_TM;
M041: NOP   0;
      A     L 0.0;
      A(;
      L     "DOOR_CLEANER_DB".BTM_SCRP_RET_OP_CT_TM;
      L     1;
      >=I;
      );
      =     "DOOR_CLEANER_DB".BTM_SCRP_RET_OP_CUT;
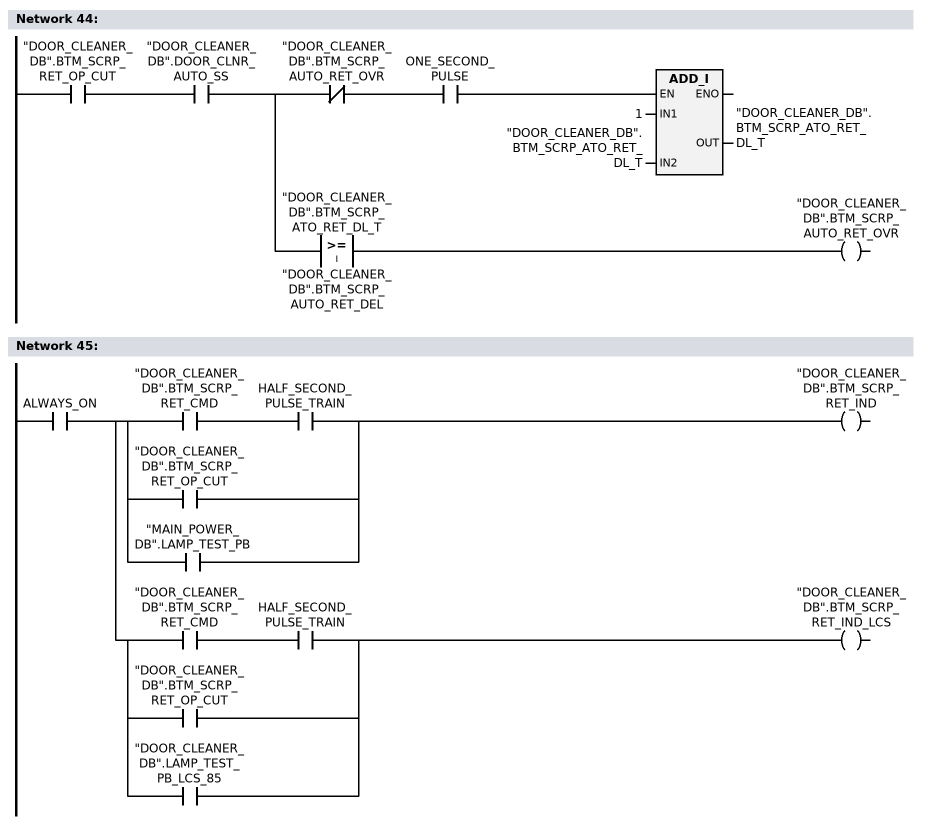
NETWORK
TITLE =
      A     "DOOR_CLEANER_DB".BTM_SCRP_RET_OP_CUT;
      A     "DOOR_CLEANER_DB".DOOR_CLNR_AUTO_SS;
      =     L 0.0;
      A     L 0.0;
      AN    "DOOR_CLEANER_DB".BTM_SCRP_AUTO_RET_OVR;
      A     "ONE_SECOND_PULSE";
      JNB   M042;
      L     1;
      L     "DOOR_CLEANER_DB".BTM_SCRP_ATO_RET_DL_T;
      +I;
      T     "DOOR_CLEANER_DB".BTM_SCRP_ATO_RET_DL_T;
M042: NOP   0;
      A     L 0.0;
      A(;
      L     "DOOR_CLEANER_DB".BTM_SCRP_ATO_RET_DL_T;
      L     "DOOR_CLEANER_DB".BTM_SCRP_AUTO_RET_DEL;
      >=I;
      );
      =     "DOOR_CLEANER_DB".BTM_SCRP_AUTO_RET_OVR;
NETWORK
TITLE =
      A     "ALWAYS_ON";
      =     L 0.0;
      A     L 0.0;
      A(;
      A     "DOOR_CLEANER_DB".BTM_SCRP_RET_CMD;
      A     "HALF_SECOND_PULSE_TRAIN";
      O     "DOOR_CLEANER_DB".BTM_SCRP_RET_OP_CUT;
      O     "MAIN_POWER_DB".LAMP_TEST_PB;
      );
      =     "DOOR_CLEANER_DB".BTM_SCRP_RET_IND;
      A     L 0.0;
      A(;
      A     "DOOR_CLEANER_DB".BTM_SCRP_RET_CMD;
      A     "HALF_SECOND_PULSE_TRAIN";
      O     "DOOR_CLEANER_DB".BTM_SCRP_RET_OP_CUT;
      O     "DOOR_CLEANER_DB".LAMP_TEST_PB_LCS_85;
      );
      =     "DOOR_CLEANER_DB".BTM_SCRP_RET_IND_LCS;
